(* CoDeSys 2.3 project: cy-wg-020-003.pro *)
(* Title: cy-wg-06 - ClevergyAS *)
(* Author: Andrea Ravasio *)
(* Libraries: Standard.lib 2.12.10 14:48:34, Util.lib 26.9.14 10:12:46, Visual.lib 2.12.10 14:48:34, WagoLibIdent.lib 25.2.13 11:12:16, WagoLibStatus.lib 2.12.10 14:48:32, SysLibFile.lib 2.12.10 14:48:34, SysLibRtc.lib 2.12.10 14:48:32, SysLibSockets.lib 10.2.11 09:20:54, SysLibEvent.lib 2.12.10 14:48:34, SysLibPlcCtrl.lib 2.12.10 14:48:32, SysLibCallback.lib 2.12.10 14:48:32, mod_com.lib 2.12.10 14:48:32, SerComm.lib 31.5.11 08:54:36, Serial_Interface_01.lib 22.4.13 12:50:14, Modb_l05.lib 22.4.13 12:50:12, Ethernet.lib 2.12.10 14:48:32, MBus_03.lib 22.7.15 16:25:47, WagoLibModbus_IP_01.lib 24.7.13 15:05:58, WagoLibMBX_01.lib 20.3.12 16:32:40, LON_01.lib 22.7.15 16:25:47 *)

(* PLC configuration (modules and I/O channels)
0750-9999/0545-0008 8 DO/DI Generic [Type_34_8_Channels] node 0, in %IB40 out %QB32 {INTTypePAAssignment = PLC; INTTypeModule = plugged}
  VPN_ST2 AT %IX20.0 [BOOLOnX_I] Ch_1 Digital input
  LAMP_AL AT %QX16.0 [BOOLOnX_Q] Ch_1 Digital output
  KEY_QE_ST AT %IX20.1 [BOOLOnX_I] Ch_2 Digital input
  EV01_OP AT %QX16.1 [BOOLOnX_Q] Ch_2 Digital output
  CTL01_ST AT %IX20.2 [BOOLOnX_I] Ch_3 Digital input
  EV01_CL AT %QX16.2 [BOOLOnX_Q] Ch_3 Digital output
  CTL02_ST AT %IX20.3 [BOOLOnX_I] Ch_4 Digital input
  EV02_OP AT %QX16.3 [BOOLOnX_Q] Ch_4 Digital output
  EV01_ST AT %IX20.4 [BOOLOnX_I] Ch_5 Digital input
  EV02_CL AT %QX16.4 [BOOLOnX_Q] Ch_5 Digital output
  EV02_ST AT %IX20.5 [BOOLOnX_I] Ch_6 Digital input
  AT %QX16.5 [BOOLOnX_Q] Ch_6 Digital output
  CIR01_AL AT %IX20.6 [BOOLOnX_I] Ch_7 Digital input
  AT %QX16.6 [BOOLOnX_Q] Ch_7 Digital output
  CIR01_AUTO AT %IX20.7 [BOOLOnX_I] Ch_8 Digital input
  AT %QX16.7 [BOOLOnX_Q] Ch_8 Digital output
0750-9999/0400-0008 8 DI Generic [Type_1_8_Channels] node 1, in %IB40 out %QB32 {INTTypePAAssignment = PLC; INTTypeModule = plugged}
  CIR02_AL AT %IX20.8 [BOOLOnX_I] I 1: Digital Input
  CIRD01_B_AL AT %IX20.9 [BOOLOnX_I] I 2: Digital Input
  CIR02_AUTO AT %IX20.10 [BOOLOnX_I] I 3: Digital Input
  CIRD01_B_AUTO AT %IX20.11 [BOOLOnX_I] I 4: Digital Input
  CIRD01_A_AL AT %IX20.12 [BOOLOnX_I] I 5: Digital Input
  CIRD02_A_AL AT %IX20.13 [BOOLOnX_I] I 6: Digital Input
  CIRD01_A_AUTO AT %IX20.14 [BOOLOnX_I] I 7: Digital Input
  CIRD02_A_AUTO AT %IX20.15 [BOOLOnX_I] I 8: Digital Input
0750-9999/0400-0008 8 DI Generic [Type_1_8_Channels] node 2, in %IB41 out %QB33 {INTTypePAAssignment = PLC; INTTypeModule = plugged}
  CIRD02_B_AL AT %IX21.0 [BOOLOnX_I] Ch_1 Digital input
  CIRD03_B_AL AT %IX21.1 [BOOLOnX_I] Ch_2 Digital input
  CIRD02_B_AUTO AT %IX21.2 [BOOLOnX_I] Ch_3 Digital input
  CIRD03_B_AUTO AT %IX21.3 [BOOLOnX_I] Ch_4 Digital input
  CIRD03_A_AL AT %IX21.4 [BOOLOnX_I] Ch_5 Digital input
  CIRD04_A_AL AT %IX21.5 [BOOLOnX_I] Ch_6 Digital input
  CIRD03_A_AUTO AT %IX21.6 [BOOLOnX_I] Ch_7 Digital input
  CIRD04_A_AUTO AT %IX21.7 [BOOLOnX_I] Ch_8 Digital input
0750-9999/0400-0008 8 DI Generic [Type_1_8_Channels] node 3, in %IB42 out %QB33 {INTTypePAAssignment = PLC; INTTypeModule = plugged}
  CIRD04_B_AL AT %IX21.8 [BOOLOnX_I] I 1: Digital Input
  CIRD05_B_AL AT %IX21.9 [BOOLOnX_I] I 2: Digital Input
  CIRD04_B_AUTO AT %IX21.10 [BOOLOnX_I] I 3: Digital Input
  CIRD05_B_AUTO AT %IX21.11 [BOOLOnX_I] I 4: Digital Input
  CIRD05_A_AL AT %IX21.12 [BOOLOnX_I] I 5: Digital Input
  CIRD06_A_AL AT %IX21.13 [BOOLOnX_I] I 6: Digital Input
  CIRD05_A_AUTO AT %IX21.14 [BOOLOnX_I] I 7: Digital Input
  CIRD06_A_AUTO AT %IX21.15 [BOOLOnX_I] I 8: Digital Input
0750-9999/0400-0004 4 DI Generic [Type_1_4_Channels] node 4, in %IB43 out %QB33 {INTTypePAAssignment = PLC; INTTypeModule = plugged}
  CIRD06_B_AL AT %IX22.0 [BOOLOnX_I] I 1: Digital Input
  ALARM_PB AT %IX22.1 [BOOLOnX_I] I 2: Digital Input
  CIRD06_B_AUTO AT %IX22.2 [BOOLOnX_I] I 3: Digital Input
  AT %IX22.3 [BOOLOnX_I] I 4: Digital Input
0753-0648 LON-FTT [Type_55_1_Channels] node 5, in %IB0 out %QB0 {INTTypePAAssignment = PLC; INTTypeModule = plugged; DataStream = 1F8B0800000000000400ED5DFB6FDAC8B7FFFD4AF77FF045BAAB560A0D06421E9B6445C134A83CB206D2ADDA0A3966006F8DCDD78FA4B97FFD3D33631B1B8F5F3C9286585A75893D3E73CECC99CF79CCF1F8F2AF5F0B957B4086A9E8DA5581FF502A704893F589A2CDAE0AB6352DF2B5C25FD7FFFD5F971D5D6B6B1632A692; DataStream = 8C387848332F7E99CA55616E59CB8BE3E3C7C7C70F8F950FBA313B2E974AFCF13FDDCE409EA385545434D392341915BCA726C94F15B85B439F19D2A20D8DCF4B17A5D2C529FC7B7251E22F4AB58B52157E14B87F94694F5AA0AB82A0A205D22CC940E38EA468CA58289D17B80152A74D5DB6C92D0B046CE80BFCFBAA509F4C; DataStream = B827DD3638995EE1E6C800067BC83674ADA5188B472075E78DCA39E96A203DA05BC99A5F151A17DF3F29D677F9A958E2CF8B8F33EE5D5782A1D1244E541E74D542AA2A7142A9FAFE7BA7DF2B705D7D62ABA8672FEE9101D40A309C1C8707B42B193FFBF7FF22D932C9B5F5ABCE45B83C448BA50A7DB427C0AD325590E1DD83; DataStream = BB78ACDA93EB528963FD7779ECDCF73D3190F525BA865BF487EFCE67F484AFE3FFF9AEB6B509FA75CD5F1ED31F1E5FC7318C794CE339BA1EB46E879A3E4154B2D583E4A6F708B369B049DF50668A26A9CCA6819BDE236DB3A3CB3FD1E4DA326C0432B87FFA1A74256D2259BAF1E4B5595DF135EB2FB11E49EAF554524DD2CC; DataStream = BBE2B5EA223CD174BAF15006FEF65A392ADBD06D503F5849179AA25E1570E705EED83720C87AD48D9F7792A148F72A32FD93B276CF772B496336D39A78CDF1B4E7BCBCAE3E3E15C237833A94A8470C5DEADD0DC7FAFDBF6303FDC746669436AD344A7B5044B769B8494069FC4D99DA944AA33268557ACD0A6B171FA15DA465; DataStream = 3A0DA344156D80B4C9505990A9F5FF196C27FD0AB4F3FDB9DE4E4432521E90AFA9FFCA9AF0B786A21B8AF5B412DEBB12683940C68322A3E113685E5DFEA9E98F2A9ACCD004B4D17727F048533100196020AFDBDAD286495D5D08B20C366FAAC8786EAE7BBA064CF8AF049A36746DAACC6C83D81458254B64580A32D707B56D; DataStream = 7A5DAD29CBFAF5C0631F9F2C3450FE0F5D572E8FBDDFBE557F1CBDEC7F5B44A8C4214265978800BE86659B2900411F382D13F1C06BF9DBC341398783F470D0B7ADD78507B583C183D3383C38DD191E4C15156117218D7BD082B6226E9AEC1E784D7788079EA22703824B32051E9CE47870B8EE015F3E1C3CA8C6E14175A778; DataStream = 90DE41C0EB1C9BFE342EC2AAED6F0F0AB51C140ED849289F1E0C2A9C87D250748468D450DA292A2CF53490404CFFAD9E26685835FDED01E1340784C3F512B2060DA13BAB8C6322CB97C7ACECF56629EDF80475918FC8501733A6A8C9A2BC530CCB96546E6A6B325D2DDCBD0A83BA9E79CE94468E59AB791E391DFEFF7E7964; DataStream = 68EE2487F9441B10269EC21278EAB0435390258314A566A4656E0BB8DFCD39F4C4CB53CA74845E2EA50CAD69A238033498E933CB3932BC226478792F3123301C4E6EF92C2E9774B6B35C9205AA8597EF62990618B0220E505AA7C14F3B4786C34286D7E7331C4E42E9EC2C0E1ACE76050D922A198B34A850C70D5362824334; DataStream = 8783C3828357E72894CF7338D8271CA4F7127244384844787D0EC22141425C56E16C6759051CF6A354C946F509E714504A4870E8E690705890F0FA9C84830104BE14E72490BBBB8184F983248F17FA24152C346FBE8C619233A4147CE47374382C74787D0E037F40F070120B0F273B4B37C29571AA5423C686BA6CE18669D3; DataStream = 8D0EED1C180E0B1872B721C785202E80BF70AB2B5AEA7D881C180E12185E9FC79023C3FE9121F718DE3C30E41EC3CBD533C5C1C2F9CE50C17C542C799E06151AAD264605414B9B7B7428E798705898903B0B39280440E1530E0A6F1E14724721DF91A08314F416F0A644BE23F1D6D1E1F5B90CF98EC41EF30B181BF2E4C29B; DataStream = 4785DC67C84121E430E4DB113930BC3E77214786FD2343EE31BC7960C83D86FCEC053A48C1B317CAF9D90B6F1E1B5E9FD3909FBDF00C672F648086FCEC85C3448657E735E4672F3CC7D90B2991213F7BE17091E1F5F90CF9D90B7B7DD93A2526E46F5A1F241CBC3A47E1905EB4FE1DE120BD979023C24122C2EB73100E0912; DataStream = 7ED3B3175242427EF6C24142C2EB73120E06107ECF4A47DFD90B299121AF743C5874787D0E435EE9F83C672FA44D37E6A50B07090CB9DB90E302FBEC851C18DE3430BC3E8F214786E7397B210786370D0CB9C790BF661D3A7B216DEE317FCDFA20312177167250089FBD9083C29B0685DC51C87724E82085CF5EC87724DE3A; DataStream = 3ABC3E9721DF917886B317F2E4C29B4685DC67C841817DF6420E0C6F1A185E9FBB9023C3F39CBD9003C39B068683F7184277CCD5AD249E2F8F3BBAD6958C9FFDFB7F81357275ED9A797DF93FDF1ACDFAB0FEEDF2AF5F0B957B408609D4AE0AFC875281439A0C03A6CDAE0AB6352DF2B5C25FD7970DC992547D767DD95254C4; DataStream = B54DF89F850C3481470A5C136EDE7924AA98066E86A7F0AA80FF85BF756321595EA31A6ED395FED50DDF7305EE56B2E65785C6C5770C5B86B420644CEEDDAFB3DAFBEF20C2171812F33BA6687E1F0CEBBD665D6C7E187EBD852709CE5D152280B0C089680AFC6A328A6D45DEC7C42F58023FE563BE725C2EF1658E3FBB2897; DataStream = 2EF872E17A1DAE092BCCABDC47C9744660002B55B6BED57E1438B28441FC0247D0F3AA705A29701896AE0A64609D2321E0DA83451FC63806120AE3C1501C35865452181A184D45A64F12AC9BC2E3F844890287B50CB35FE0469A029DFDA15A7FB6B5074955269C691930B1D08DA9DB868CFE98597FB285F2B12F68F68273C9; DataStream = 63EEC6169EBB5FCAC25E10510064E8EF22EF0A2346CB21F4465D96149EE80365A6398AE588E24A32F50D11A7C1536681C3DC21BA189C213DC1A09820D34833492FA05333980BB3AD5968860CD257DB1CC8F81D1AF2C74ACE9393CA892B1EE98925DCA837687FEA09CD71A7DFFB54E0FAD3A9892C42282CB04289E0CE50DD27; DataStream = 6E3920AED36ADF123990CEE1578C759B397111B255D89349C88D3D72D1522E1455554C24EBDAC44C2527CCF4B7CA6A2D790BA8095A01561E6B02274D26A0E3265B8C76BFB762FF84C5FE046BB94783327CE232ECE290D749CAF55F5EF15C7679AE53129C851F03E0B58CA7B8B51FCB3466C772B9ADB8DCB27A48AB4B83B98E; DataStream = 29A651A64AC58703954A483E620462746A70D3179304A444429AE4C1C359F15EB138DB619E03C4A30ED27E574E7080958CC850DB0819F85A94A8EB8E0371A336B14F8E69B1EF356415357D82E2D6542AFD34B5E8A56432FAD98396F23E25E55F938E7E542C6F72D60472C04F5F488AC662FF637BD84AD0B789F37034DBDE44; DataStream = D1A699AD1277CA1111E01F9F4D74043AF50B543E7545EA81326C2890461E8D1687E8994622AD2C42544342543D21AA7E217C6615F09693719364514ED99694D884185988189C3EE5705305A533A21B4B343424CD9448C8439C052359AE33E642F935761E8F168D3480D183C9CA0AE61940A17C721284BB2C2070CE443A874C; DataStream = B464B4855F05B700EED31FFEA54459F864E8F6726BC89E2DA3217B16E8616B004B42E1A04A6D84BDF7BAAE2249DB076CD5562A047D6EC8BF491E4D01C274E869F3376F3A281F23CD36A1ED5441EA6443516C42224E94A4483A3725B9290900F0D6966446A96CA7926CD3B289C1D9CCE57600DEB6E6785340A611BACE449CA8; DataStream = C1E14BCC8817488EF558F4C98EF99BC8E6E6B8B34AC5CC0B2D815806A9B6701CAA3FFC2BD4CD48560319497A12E5A60949F769277E3DDD7D4E92F6104849F23C3327398894242A25B9E23E3623499B4527246BFB4F42F43CE4C61C45E4BDD2A726A92118EBD3B1432E3A15E118A47D0B38402A922D62E1D5F8283D4576D274; DataStream = 888D29B19D656071663226CBB76936529A181E673BCBEA3B10109148950D6569E94C839C2A7098F848EC9AF3BA61484FDFF8DA0FACEE2D3A43539D93F0650ED1ADD295C78BB75A4CF2880FAFBDA75802D645B1FE35413E023D9480830835573CCA07B0C6D738792E19E0E02023459298AC8E063C90D2F66030F5A15CF92C24; DataStream = DCFA9030E6922E99C64D5D5C095C66DA5A4FE26FFCC98FB53513858E34D9551F34DAEDD5506C6EB4483F7FDBD224A533C6574FAB67955AF53429367386E1EF51BDE91B0626323262B435E9AB9E917EB23279D01B22E330296D1904C47296D039F59ADDA92392089AA9B7437CDB37E7BB851F8A3E3474E6DACD08F461828FF7; DataStream = D0A6E04303E9B13271650B634F8DA3DAB7DF182752FC6D1D7B4FC26F21AC49974D7FA6E0A6B636122AD266D67CFB10C091DF25173D00428FE3ABE7A5B322EFA657DC677EBB4C292E48D84DAA74F7715CF2A643A4544C0733EBFE4396087D0B98E57D5B7CFCAA06E5ACE20F9110F700CE71BCEF1711F2916306199B95D88556; DataStream = 1E94892DA91C5EB0649DEE20674CD9C5144BD1A9A330AFF04069373983E8C46402BF7C467EF9FDF05B4ECB6F3923BFE5FDF05B49CB6F2523BF95FDF05B4DCB6F3523BFD5FDF07B9296DF938CFC9EEC87DF5A5A7E6B19F9ADED87DFD3B4FC9E66E4F77487FCA6E3F02C3959CF746DE0D9B31706DFF3CD593F7F611CE6630C5D; DataStream = 12EFFC9E8C5E6A50E663AC5E22F37BB280A9119A8F318189CCEFC91CA6866B3EC61E2632BF27DB981ABBF918E398C8FC9E0C656A20E7632C6522F3A9ADE6CEAAFEDC88C0CBC2E082788E7C7268837860F5BD22977B6F03E80949C611B7D0356B7EC44DA4A7236EAEDBF88AA2D9163AE2684170CAAC69FACC59A584ABFC199B; DataStream = 435F91C48E78FC39B4B0984FE4B1B87460D92F71967460A6F8D515A38B07344BFCCA0CCA17944AB4EE91067B12A6B24A9449CC62E828519891F8448AAD7880DB7B12A3EC05D537A0D859E4A8B2E4981322D182E0FB7B92E4E4DCD32EB238B7AE915D386462F48BB4D8BB3C030A3219E461160E39581597C3F2BDDEB04DFEC6; DataStream = 9727E7573BF667DED60FF952CCE65BF6E4CB311E70ED2563DED19DFA8F0C0973F799987C795820D57BE86573E451026FB9865CF1B225C8B1C05BE7C737DCA7A2AF1E466C7B64793B422784E8F647E486156D947AEF9ED49310F51FE3ADB0403949A51CF0182AC1C566456CBFD19A92D8BAB5557F719BA892D74D7485C9695A; DataStream = 11974EA1D258450F484D5335E39536912792256596B105BB8D937619E82E5AE2B3677AC90F0345EF2E4B3D0D73438BE8E1D8D2C71867E3F4565975CAC9926D62B0756039515E8AB35582B37738C51E01B25516C8DED1BDB3C41D49F6368EB3F3B6B603EE416DF559A096297386AD1C26D012C948994C4C28F6BCB04A8398F8; DataStream = B8254A3B9988CA88625E41E8C23341F575C62E3C13365F61F0C22E1E7AA5D10BBB04E815872F65F61E7CA6F865D768767EEE9B21EF55F02C154DCCC07FE1A7B5B3B7CFFD2696FA7FAAB2000F3B83A1F53D96C2DCB2CBB5A8E7E8D07859A31B330A19F432C63F26A4B733C05B84DCC1725EC7F93CF7CC2FA9B55CEAA612159F; DataStream = A6299287E74351EA129F7F868C23B79E67FFC591229226C75FC0F7C60291CE134B2519AF183D8E97564246D4D354525D8DA76EF59EE2FE8FB9F0844C51AB15C419665E0E048EACD2F24066F55ED5AA2674E73AE939524EA0BDF95132103B8F7DA7B1048E9368378F3CCABF51C2E019B3040E61D65938E52A33844E9E906008; DataStream = CD34D2C16EE342683DD05D74088D23D52D15D1B779545EED1E9D57D624DF3821893531F80A51CDAF88CE8B3753559AA5377307A38D89C51A4ECEB6D86E92214ADE88642A9E42A9B079DFC1562A9F4E08579D7720C96A0D3D7F294753313191C936724C1C1A2F52CED1B7ADA23E2D12AFCCDC460ADDB6F00B6694D08B1477F4; DataStream = 97482BCA8A21DBCA567AA5039DB143E7450A3D9C3931E9C9893B981487D28B147E74913C9734053A2E4E255BDD6A66161EAD31A1F522C5202D8426F792FC13C45154DBD86A7EA60EADB143EB99CAFEFA0FC8281A92364BCB3C3324D781CA985079114B3202BBBA03296C4C669F6224581001BFBB6A645E1F4C5990476B9FEB; DataStream = 23C1A28C344CA368E9C50592CCF40B2462763031BCD3E2107B11CBD2D0170B5B738E3A30332E7CA65C3250DCC3A24F6F635AD0379A808D51A7452BBD23C61406CB31C694C6D6DEFCB0A4F242578EA2A2159798437CF8D0163279E28C156DEC127C117B434F222E8229DF461E955019B30FEFDC878DE94A9A0D9826EB9A65E8; DataStream = 6A4AD699399905A1347628BD50D4B2049F8C6EDD6F2109A8925B93F3FC8686CA808DB6A14CD2825794182E9917B130225AEA86555C48E6CF6DC43008993126F32256C5E548D16645FC81AC6D6459AE68918F6DBD884DF10B846DC2AE04C2B45EC4AA90CD90A2A65BCAF4A938C916EA33A5A25B2094E078BF717F82551191C9; DataStream = 7EDF37D5C2817B80C78BA58AE2774E3738A2EF8CF39B16AF1412F7693CA0498AD736985B6CBEE7F771FAD61689FED53BD8E4239A1BA4554DE7C1B5FC232975A15955B4975DC355D94A64B5D1FA0E6174A9913329EE3B121F69C67D6D82FE971C8964ABAA5BBE96A857836DCE140E1E361577D6C87AFD47D4F15309878D7882; DataStream = 92B6E47CBB2DCF5771D2E3EE16C149CAC297F2692D701E4DF9B4C27B5B8BF8932D78EF81C42E99DFB1F07DCA253818EEB497E35EBB9820F0C491C935906A2A769A2D46B2CB43BE4269F906E22CA0C8CC39BFB9AB37B845C4010251678C05BF791937C51EF9982D9D6AE4EC9BD797BEF6C1BFB8D5971386D2CC39EB67B5C175; DataStream = 7D492BEB020979CE59C261895AE2B837EA1438517A246DE8101D07A90C3075CD522495936419C75E06C27BD74C72FD5BA1371EF6C703A1D74C41E911EFEF2690128586D0BE13FC5C86996CA8BA8938490370971E9073F418936CA3D31F08E356BB13A0588EA13841D81626D36C0A1D6118265D099116C9919DC0E6847C9246; DataStream = 379EDCEF0930A937DB3004C3BEF815D65DFFF3E8D64FBC1A260E2CEB8B8C533516EB7EAA270954334CDB1A657AC0DEB14FA399EA5DF3ABB7776E6056ED1EA4D06E521662E1E34DA7C8E04C9B0808662882E03F2D0144FC1C22D3F46652D5F59FF8C8DF244A742E09AD38C5160C4337387C0AE71269D86B8954C3011DFA56BD; DataStream = DD89D76C8FE4648DE9784E05518C57EBE0502A1AB7CAAD448FE5A8D714C42FB88E2A4EA93D96B13EC3281C630D4C188D767F9DE5B05A0759C62F414E38924761521CB6BB427F345C275B0B91FDA2C06A79E44C827732E210663F82E89776AFD9FFB24EF3344473ED50562FC1C8245A1F0D6FD6499E8549D2D54C0D956E81CE; DataStream = 2E71D88CD88801541B0D61308029ABDFAD29D9790260DCA3271D9054E8334F4500D20341F83C6EF7EEEA1DBC6DEF5B10A5F09C39ADBFD4DB4CAF3378DF478A4F873DA70EF604DE3109B2305A4EB00FE7CDEF1CB4123127B8DE19DF087550F1200C8517CF3AC9A9AE5B91245BFDFE709D64789D37D1BD3D23C70BE20F7A6109; DataStream = DFE1599634FA9AC2FB08E24DE1E3E85390761896DA3EAA36653D15F176AFD50FD20E4FF0E0C9041F323BE383AF83A1D00D77115E9FC3B973B634A7989C536B104114347224B034B31846930059095C7C0D4C97E61CA2944E8646BF87BF961650DC62180F714F1344B690A12B7D3A55158D890540B2DF6A75DABD804B520CEB; DataStream = 1F2D0EC5C5B50A9D540D7FE90F467E213DC1F2E526D0D2D28954BE0D1317863840E7B9644C1E25BC7742AF458938EA7DEEF5BFF402FC8495D7B5EEBE77AA9C6194D63825C8B54432FE86E524AAD36447A0A773EB949738B3A031AD0126D9C7B3D56C0FC9B1B0EBCB59F358CA48B6DEE9FAE9C6F90643DD92D463B796801482; DataStream = 3E60DF9AF4C773EF701A47D7A02B526106C6DEE4DCC6305FF80C3A0B6912A04DD4A80DFBC3F1E0AE4178E2E39D8A585E981BE46BF4CBF1CE452C7DE6B6C81AFD4ABC87E1144783D5760AA4E9A4A948323866C80FE43B60B73BDD21B8FF627078C2D010473E6A74FCE4CBF10E07253F5766F30CECDFB43FDDB0F967781F711D; DataStream = 440910E8A09CE08B30072869E4438A197644D88493C63CA4910C3B15312689C31D629A615F2368278E7498EFF0526D0112AC835294A3D11631C9004196E30F0401D58AE989DE8A428870785162C24503E18F0D4FC04DD7ED7B70D7DF91FA87F7A9BA198A1F03B8CFB342005F1FE00163843175F2FD0E17B0DFA10FB30F4760; DataStream = 640C45FBA942A08011DC8C3171B8EBC1E8F62ED07578D506C5C33BDCC4154F3F8A4361300C0D6378F146F4936DC6485FAC690BAFE5407F0B9A8AE390F6A018BA86DF3701DCC6A60969267522E80BC410DAC97376ECE1B020F4EE1AFDEEEDB85BFF27C04178D1073890EE35EC48AA603596B6954AD86EBFD71EF64562880376; DataStream = 8F118E0485F56C2A4C2332A28C3CE9A3DEEEE1D913C480B75766E428F0177D3969B9545DB72B32A0C4B4EB43F81782BF7E305E0FB3DE8788D2A0B41247254C2FCC27A5073E2049542451FC52177BED5E20D2A894D38568674E88167A473E6386E8364DFEB3A33FE2221ABA52966BEFD8336976843BA1330E8FB7778B6922FC; DataStream = 77E3BC3EAF1DD318F8EFC6F96B37605A3612AB12EFA7759429E206D21401316217882533B9771FEB0D7C38B077484199099EB76B9E48D826DCD2EF683FA5EAA412D54939DE5D2344073E6340ED71887E358A7E25DE5F23F487D4A01DB7486DE0BBA6622E55E9E97DB89793A85EAAF14E1BE9E516E089707FC4916D8906CE9C; DataStream = C980270284044B0CC751C2D5A2BAADC5BB72A49BA819398B227A16EFC645F12E0E7B475407E057DC20F2A548852B25387AA46F425EA558E02E17563791A3C6D7183E5F22D4617608D6855E66CA8875E2DF29B04E203599CE8B5364F3C3400BFD01AE7845416CCA7DB15BEF30B2E2A68F5EC4B3CDF6A0FEB12334E3518F1606; DataStream = B99CB96F1A31098E6E9BF521DE59AF0F47837814BC45064E327964DD52C308CA03A1D3228E503C063AB93C2970C4531CABF54E5DECC6C39E23BFF31E153E2A88163731C98AC26D5F1C828731F81C8F737DB7642C7686FA7760FDDB4D211ED302BA134149E8E1A98E472DD1D1383A25098A2776EF98EC8551A94142D534FAD3; DataStream = E8087591A13E61500AD074CAFF624886A6998135CE2852DD21D5448A7B3A169332A109EB6FD86E7D7586B7C9C019D6AADCAC0FE672656C320590644AF24DB8D693F36A3D995D75EBBD114E830EC560DC165E64E10E305491CA8AB80E44A1DB871517EA80B1E7443BF055ABE10A1592D6A3624C9599ED80F5923A25E43B8CCC; DataStream = 6E6FC5FE27B11E9CFCF072A4FA446AB08A6E0D16A949E3DE050BB39836C6D333511808C1AD0FC66AFD85641BA8D3CEBC6D0790307601874987173095022050E2547D16CB69A71FF0FF19B164479720669D7BF3B04AF5E21DC641E376886FD06F8E4574D5E9D79BCC0960EC5AD91AE94CB60D03BC0B15EF8C4A13E8CBE9FD03; DataStream = D79E06B879944C6E2EA934F6C3FAAD3E1D4103C5E41E1515C7B4265874CEB035BA776BE80BFA387E6D1FA7EE57CF7F881AF1518FC53C2312BD013A09DC0F3DCE964ED55C706C49691236FB12FECE3BD50AF0B1605470DA1FDFF08BE57F9488F608F11FE2C036258B7553EF0C9972B14C3FF065C48BB61ADA7B3453C868470E; DataStream = 28D8EFBAC8EE3C8C63234D753530AAEF28DBDE8B52BC3203CDE8723449471AFA65E1A5435C5D7DE97A84EFF0268F53F4877DDF23580126293F84BB47F401EE1EBF0D70C4214BFEF01EAFE6247D589FFC850DFEED3DE2FEF88FAD5B7F2A1315D15F78C780FEA2F3EA5CC55B42B28C9616557A474B8E381DA7021E15936A03D6; DataStream = 19A0A9CC34DD009508746B20CB3634135362D07734726AE144051923F245D269A0BB286F6D28DC3287BF9AD2F5AE3AAEB75361C676B81FA21C6E1C35A470B91BD45CE1B4A2645B3A218061047F864D9B21BC776E3D22A405F23F387FC73435A4D3FA68D80FA3039248C584AEA9CC4223F2E48D501FC6FBE1F5151745078A65; DataStream = 6087A67C1E714D35BB8E8490EF8ABD4FE32F623758C3C4A8BDD2753591D746BFDF89F7C399BC6ACA6C0E119C6DCC6266ADFDE9060062247E12E2BD72660F38AF2AEB6C0F8490C759D475EE19CEC04A31F016A7E3D6D071B1ADA56D452B40BFD54AF0D5BDF8F91E618238E661A75E09BDF590276CF305583C33F0209E702D84; DataStream = 454B4ADE919F4B7BB164BA2B84B2D015C44F21B5636C0F29DE28D0A4220290994A60AD013C70D10ED377255DB4EABD71BFD7F99AE0CA3B2AF7A85873929DC6297E9D76EA98EFE81E44213CA10CDFBE2DA3E242FA89BBA115A411F4DA0D21C18577EA5BC9602792EBD6FF092F6C86C70E63AB2F407F31521CE3F188272B34FA; DataStream = BD7EF76B829BDE44737BA14CBC10239E6653B81975D72A80C2ABAE01C07B6FA420D7A877DA1F4588B013FCEE95F6CAC962138D0DCD36638D7944616D81A14B41152C563D6933C79B52CA42CC9C877864A7EAC637770DE223475B05AF41ACF34CA1B31F4FCBBB1F726583F6F83858027D8C2BF5AE2F49BD5EDB84FF8143E0D4; DataStream = 5E3721D0B84386090DB1B67C006AB8192DEA6E2D212A68913A22AFCD096ED295FED50DDF63C0B064CD41B72EBE3B9C132A26F7EED759EDFDF78EAE7DD18D9FE67752A0FD1DD7E834EB62F343EBD6A9416B0333A512C7FA0F6445536017E2ABD856F8030E03FC0906BC3C8FF9CA71B9C49739FEECA25CBA80F50AD2DB1AF1F5; DataStream = 24157A249F7B665CF3BC17B7D61D7F278FEB7B419DA2C9CA5252234E2D188040F893774EFB50013E0C7E173C2E09578DD2F70A103E308B7ED4DAD7E9FA414AE19EB4074574EFE241F51D8E15AEFB4FE876FD40ADE8F48EF6A0BB1F17F7775A61761AECC47B99872861BC64B8094817E8E4344D27B54027B172E01658966027; DataStream = D5149D9C063A599D891729CAADBE365ECE8A0D291FEBDA6AF51E37F046A63EBBFEF103FEE8E0772160194F25195DFF3F0534515341320100; DataStream = .; DataStream = .; DataStream = .; DataStream = .; DataStream = .; DataStream = .; DataStream = .; DataStream = .; DataStream = .; DataStream = .; DataStream = .; DataStream = .; DataStream = .; DataStream = .; DataStream = .; DataStream = .; DataStream = .; DataStream = .; DataStream = .; DataStream = .; DataStream = .; DataStream = .; DataStream = .; DataStream = .; DataStream = .; DataStream = .; DataStream = .; DataStream = .; DataStream = .; DataStream = .; DataStream = .; DataStream = .; DataStream = .; DataStream = .; DataStream = .; DataStream = .; DataStream = .; DataStream = .; DataStream = .; DataStream = .; DataStream = .; DataStream = .; DataStream = .; DataStream = .; DataStream = .; DataStream = .; DataStream = .; DataStream = .; DataStream = .; DataStream = .; DataStream = .; DataStream = .; DataStream = .; DataStream = .; DataStream = .; DataStream = .; DataStream = .; DataStream = .; DataStream = .; DataStream = .; DataStream = .; DataStream = .; DataStream = .; DataStream = .; DataStream = .; DataStream = .; DataStream = .; DataStream = .; DataStream = .; DataStream = .; DataStream = .; DataStream = .; DataStream = .; DataStream = .; DataStream = .; DataStream = .; DataStream = .; DataStream = .; DataStream = .; DataStream = .; DataStream = .; DataStream = .; DataStream = .; DataStream = .; DataStream = .; DataStream = .; DataStream = .; DataStream = .; DataStream = .; DataStream = .; DataStream = .; DataStream = .; DataStream = .; DataStream = .; DataStream = .; DataStream = .; DataStream = .; DataStream = .; DataStream = .; DataStream = .; DataStream = .; DataStream = .; DataStream = .; DataStream = .; DataStream = .; DataStream = .; DataStream = .; DataStream = .; DataStream = .; DataStream = .; DataStream = .; DataStream = .; DataStream = .; DataStream = .; DataStream = .; DataStream = .; DataStream = .; DataStream = .; DataStream = .; DataStream = .; DataStream = .; DataStream = .; DataStream = .; DataStream = .; DataStream = .; DataStream = .; DataStream = .; DataStream = .; DataStream = .; DataStream = .; DataStream = .; DataStream = .; DataStream = .; DataStream = .; DataStream = .; DataStream = .; DataStream = .; DataStream = .}
  AT %IB0 [BYTEOnB_I] First Byte of 24
  AT %QB0 [BYTEOnB_Q] First Byte of 24
0750-0464#04 2/4 AI RTD / ADJ./ HA [Type_44_4_Channels] node 6, in %IB36 out %QB28 {INTTypePAAssignment = PLC; INTTypeModule = plugged}
  S01 AT %IW12 [INTOnW_I] Channel 1
  S02 AT %IW13 [INTOnW_I] Channel 2
  S03 AT %IW14 [INTOnW_I] Channel 3
  AT %IW15 [INTOnW_I] Channel 4
0750-0650/0003-0000#03 RS 232 C Interface (Adjustable), 3 Byte [Type_21_1_Channels] node 7, in %IB60 out %QB52 {INTTypePAAssignment = PLC; INTTypeModule = plugged}
  AT %IX16.0 [BOOLOnX_I] Transmission acknowledgement
  AT %IX16.1 [BOOLOnX_I] Reception request
  AT %IX16.2 [BOOLOnX_I] Initialization acknowledgement
  AT %IX16.3 [BOOLOnX_I] Input buffer is full
  AT %IX16.4 [BOOLOnX_I] Number of received characters Bit 0
  AT %IX16.5 [BOOLOnX_I] Number of received characters Bit 1
  AT %IX16.6 [BOOLOnX_I] Number of received characters Bit 2
  AT %IB33 [BYTEOnB_I] Input data Byte 0
  AT %IB34 [BYTEOnB_I] Input data Byte 1
  AT %IB35 [BYTEOnB_I] Input data Byte 2
  AT %QX12.0 [BOOLOnX_Q] Transmission request
  AT %QX12.1 [BOOLOnX_Q] Reception acknowledgement
  AT %QX12.2 [BOOLOnX_Q] Initialization request
  AT %QX12.4 [BOOLOnX_Q] Number of characters Bit 0
  AT %QX12.5 [BOOLOnX_Q] Number of characters Bit 1
  AT %QX12.6 [BOOLOnX_Q] Number of characters Bit 2
  AT %QB25 [BYTEOnB_Q] Output data Byte 0
  AT %QB26 [BYTEOnB_Q] Output data Byte 1
  AT %QB27 [BYTEOnB_Q] Output data Byte 2
0750-0653/0003-0000#03 RS485 Interface (Adjustable), 3 Bytes [Type_21_1_Channels] node 8, in %IB68 out %QB52 {INTTypePAAssignment = PLC; INTTypeModule = plugged}
  AT %IX18.0 [BOOLOnX_I] Transmission acknowledgement
  AT %IX18.1 [BOOLOnX_I] Reception request
  AT %IX18.2 [BOOLOnX_I] Initialization acknowledgement
  AT %IX18.3 [BOOLOnX_I] Input buffer is full
  AT %IX18.4 [BOOLOnX_I] Number of received characters Bit 0
  AT %IX18.5 [BOOLOnX_I] Number of received characters Bit 1
  AT %IX18.6 [BOOLOnX_I] Number of received characters Bit 2
  AT %IB37 [BYTEOnB_I] Input data Byte 0
  AT %IB38 [BYTEOnB_I] Input data Byte 1
  AT %IB39 [BYTEOnB_I] Input data Byte 2
  AT %QX14.0 [BOOLOnX_Q] Transmission request
  AT %QX14.1 [BOOLOnX_Q] Reception acknowledgement
  AT %QX14.2 [BOOLOnX_Q] Initialization request
  AT %QX14.4 [BOOLOnX_Q] Number of characters Bit 0
  AT %QX14.5 [BOOLOnX_Q] Number of characters Bit 1
  AT %QX14.6 [BOOLOnX_Q] Number of characters Bit 2
  AT %QB29 [BYTEOnB_Q] Output data Byte 0
  AT %QB30 [BYTEOnB_Q] Output data Byte 1
  AT %QB31 [BYTEOnB_Q] Output data Byte 2
Fieldbus variables [FB_VARS] node 1, in %IB0 out %QB0
Flag variables [FLAG_VARS] node 2, in %IB0 out %QB0
Modbus-Master [MB_MASTER] node 3, in %IB0 out %QB0
*)

(* Global variable list: Global_Constants *)
VAR_GLOBAL CONSTANT

	Plant_NAME			: STRING :='cySN:20 cyVER:1 - ';
	Plant_SN			: DWORD  :=20;	(* S/N Impianto di telecontrollo *)
	Plant_SW_VER		: WORD   :=1;		(* Versione SW installata *)


	(* Colour defines *)
	COLOR_RED			: DWORD	:= 16#2020F0;
	COLOR_YELLOW		: DWORD	:= 16#20F0F0;
	COLOR_GREEN			: DWORD	:= 16#20F020;
	COLOR_LIGHT_GREEN	: DWORD := 16#006000;

	(* Parameters *)
	Plant_DefaultTAmb	: INT	:=100;		(* [.1°C] Temperatura ambiente di default in caso di rottura sonda *)
	Plant_MaxRunTAmb	: INT   :=250; 		(* [.1°C] Temperatura ambiente massima funzionamento impianto *)
	Plant_AntiFreezeTAmb: INT   :=-40;		(* [.1°C] Antifreeze temperature, start circulators *)
	Plant_VRD_TAlarm	: INT   :=450; 		(* [.1°C] Temperatura di allarme VRD, blocco *)
	Plant_VRD_TMax		: INT   :=430; 		(* [.1°C] Setpoint massimo per uscita VRD *)
	Plant_VRD_TDefault	: INT	:=300;		(* [.1°C] Temperatura di default in caso di errore climatica *)
	Plant_CirOffDelay	: TIME	:=T#30m;	(* (Def.T#15m) Ritardo spegnimento pompe per ricircolo caldaia *)
	Plant_CirOnDelay	: TIME	:=T#15m;
	Plant_MaxWaterLoss	: WORD  :=2;		(* [lt/h] Massima perdita del circuito *)

	(* Filesystem *)
	FilesPath  			: STRING :='S:\';

	(* TCP Logger *)
	Logger_SERVER		: STRING:='';
	Logger_IP			: STRING:='192.168.100.3';
	Logger_PORT			: WORD  :=80;
	Logger_GETSTART		: STRING:='GET /cygmsrv/hsgm.ashx?';
	Logger_GETEND		: STRING:='$R$N$R$N';
	Logger_CHECK		: STRING:='True';
	Logger_CRLF			: STRING:='$R$N';
	Logger_DataFile		: STRING:='S:\LOG.DAT';
	Logger_DataFileOld	: STRING:='S:\LOG.BCK';
	Logger_IndexFile	: STRING:='S:\LOG.IDX';
	Logger_ConnRetries	: BYTE:=5;
	Logger_RecoverMsgs	: BYTE:=25;

	(* TCP Remote *)
	Remote_PORT			: WORD  :=10;
	Remote_WELCOME		: STRING:='Connected$R$N';
	Remote_OK			: STRING:='OK$R$N';
	Remote_ERROR		: STRING:='ERROR$R$N';

	(* TCP Sockets *)
	MAX_SEND_TCP_SERVER					 : DWORD:=3000;(*60000*)
	MAX_RECEIVE_TCP_SERVER				 : DWORD:=3000;
	MAX_RECEIVE_TCP_SERVER_SOCKET	 	 : DWORD:=1500;
	MAX_SEND_TCP_CLIENT					 : DWORD:=3000;(*15000*)
	MAX_RECEIVE_TCP_CLIENT				 : DWORD:=1500;
	MAX_RECEIVE_TCP_CLIENT_SOCKET		 : DWORD:=1500;
	MAX_RECEIVE_UDP_SERVER				 : INT  :=1472;
	MAX_RECEIVE_UDP_CLIENT				 : INT  :=1472;
	CONNECT_WATCHDOG_TIME				 : TIME :=t#10s;

END_VAR

(* Global variable list: Global_Retain *)
VAR_GLOBAL RETAIN PERSISTENT
	Mode_Manual : BOOL := FALSE;

	CAL01_Clima : typ_Clima;
	CAL02_Clima : typ_Clima;

	VRD01_Clima : typ_Clima;
	VRD02_Clima : typ_Clima;

	Ctl01_Counter	:	DWORD;	(* Water counter *)
	Ctl02_Counter	:	DWORD;
END_VAR

(* Global variable list: Global_Variables *)
VAR_GLOBAL

	SYS    : typ_SYS;
	Logger : typ_Logger;

	Lamp	:	PLANT_STATUS;
	T_AMB	:	INT;		(* Environment temperature *)

	(**** PLANT OBJECTS ****)
	(*...*)
	(* Boiler *)
	CAL01	:	obj_CAL_VT100GC1B := (ID:=1);
	CAL02	:	obj_CAL_VT100GC1B := (ID:=2);

	(* Cascade *)
	CAS01	:	obj_CASCADE	:= (Tmonitor_On:=T#45m, Tmonitor_Off:=T#30m, DeltaTempThr:=70);

	(* Water counter (NB: weight is multiplied by 10) *)
	CTL01	:	obj_CTL	:= (ID:=1, Peso:=25);	(* Domestic water	-	2.5 mc/h --- 2 impulsi/litro *)
	CTL02	:	obj_CTL	:= (ID:=2, Peso:=25);	(* Compensation		-	2.5	mc/h --- 2 impulsi/litro *)

	(* Heat counter *)
	CTB01	:	obj_MBUS_CTB_SHARKY775 := (ID:=1, Address:=16#51865849);

	(* Cronothermostat *)
	THER01	:	obj_CRONTER := (ID:=1, Local_MaxRunTAmb:=250);
	THER02	:	obj_CRONTER := (ID:=2, Local_MaxRunTAmb:=250);
	THER03	:	obj_CRONTER := (ID:=3, Local_MaxRunTAmb:=250);
	THER04	:	obj_CRONTER := (ID:=4, Local_MaxRunTAmb:=250);
	THER05	:	obj_CRONTER := (ID:=5, Local_MaxRunTAmb:=250);
	THER06	:	obj_CRONTER := (ID:=6, Local_MaxRunTAmb:=250);

	CronEd	: 	obj_CRON_EDITOR;

	(* Pumps *)
	CIR01	:	obj_MODBUS_CIR := (ID:=1, Address:=1, OnDelay:=T#1m, OffDelay:=T#30m);
	CIR02	:	obj_MODBUS_CIR := (ID:=2, Address:=2, OnDelay:=T#1m, OffDelay:=T#30m);

	(* Double pumps *)
	CIRD01	:	obj_MODBUS_CIR_DOPPIO_new := (ID:=1, Address1:=3, Address2:=4, OnDelay:=T#1m, OffDelay:=T#10m, Mode:=1);
	CIRD02	:	obj_MODBUS_CIR_DOPPIO_new := (ID:=2, Address1:=5, Address2:=6, OnDelay:=T#1m, OffDelay:=T#10m, Mode:=1);
	CIRD03	:	obj_MODBUS_CIR_DOPPIO_new := (ID:=3, Address1:=7, Address2:=8, OnDelay:=T#1m, OffDelay:=T#10m, Mode:=1);
	CIRD04	:	obj_MODBUS_CIR_DOPPIO_new := (ID:=4, Address1:=9, Address2:=10, OnDelay:=T#1m, OffDelay:=T#10m, Mode:=1);
	CIRD05	:	obj_MODBUS_CIR_DOPPIO_new := (ID:=5, Address1:=11, Address2:=12, OnDelay:=T#1m, OffDelay:=T#10m, Mode:=1);
	CIRD06	:	obj_MODBUS_CIR_DOPPIO_new := (ID:=6, Address1:=13, Address2:=14, OnDelay:=T#1m, OffDelay:=T#10m, Mode:=1);

	(* Temperature probes *)
	TPV01	:	obj_TPV := (ID:=1);
	TPV02	:	obj_TPV := (ID:=2, IN_WMIN:=50 , IN_WMAX:=800);
	TPV03	:	obj_TPV := (ID:=3, IN_WMIN:=50 , IN_WMAX:=800);

	(* Zigbee temperature probes *)
	ZTHL04	:	obj_ZTHL := (ID:=1, Address:=1);
	ZTHL05	:	obj_ZTHL := (ID:=2, Address:=2);
	ZTHL06	:	obj_ZTHL := (ID:=3, Address:=3);
	ZTHL07	:	obj_ZTHL := (ID:=4, Address:=4);
	ZTHL08	:	obj_ZTHL := (ID:=5, Address:=5);
	ZTHL09	:	obj_ZTHL := (ID:=6, Address:=6);
	ZTHL10	:	obj_ZTHL := (ID:=7, Address:=7);
	ZTHL11	:	obj_ZTHL := (ID:=8, Address:=8);

	(** Communication **)
	(* ModBus *)
	MODB01	:	obj_MODBUS		:= (ID:=1, COM:=3, BAUDRATE:=BAUD_19200, RS485:=TRUE);
	MODB02	:	obj_MODBUS_TCP 	:= (ID:=1, IP:='192.168.100.11');

	(* M-Bus *)
	MBUS01	:	obj_MBUS		:= (ID:=1, COM:=2, BAUDRATE:=BAUD_2400);

	(**** SIMULATION ONLY ****)
	(*...*)
END_VAR

(* Global variable list: LON/Module_1/InterfaceBlock_Module_1 *)
VAR_GLOBAL CONSTANT
(******************************************)
(* Automatic generated code, do not edit! *)
(******************************************)
	abSignature_Module_1 : ARRAY[0..15] OF BYTE := 16#67,16#E5,16#C2,16#E0,16#43,16#BD,16#55,16#4D,16#BE,16#30,16#A9,16#FE,16#D9,16#26,16#7B,16#E7;
	wConfigSize_Module_1 : WORD := 522;
	abInterface_Module_1 : ARRAY[0..130] OF DWORD :=
		16#302841AA, 16#214BDC0F, 16#6041B800, 16#06246830, 16#428B2E71, 16#64B95263, 16#FE000902, 16#2A050140, 
		16#0028C092, 16#037C10FF, 16#6D81026F, 16#0418B0E4, 16#C75C1D07, 16#9CD47157, 16#5A1D2B75, 16#1D531D1E, 
		16#4F0D2658, 16#5AC76C1D, 16#2D5F874A, 16#FE884D09, 16#CE34C958, 16#4CA0345D, 16#856A742A, 16#B26FDD52, 
		16#2BF66959, 16#74C79655, 16#966CD09D, 16#DFE60549, 16#2C48B975, 16#B66DFB76, 16#48BA6ECB, 16#955B162D, 
		16#B7300196, 16#2B35AD5D, 16#65EBC62D, 16#2106DDB9, 16#564CBE30, 16#DDA96F05, 16#AD4B372C, 16#255378CD, 
		16#36ADD181, 16#59D42ACB, 16#9B603585, 16#DDC49858, 16#EA45B329, 16#CD59F616, 16#B50A12E0, 16#56B5BE52, 
		16#8C890100, 16#5AAA1481, 16#B253E154, 16#6C831684, 16#A2ADDCB0, 16#4ABD13A9, 16#950B79D9, 16#4A948694, 
		16#4DBF5E45, 16#CA018948, 16#054C41E5, 16#B86DCB52, 16#2FBEA018, 16#40AAB4D0, 16#A1F866E7, 16#E288A8D1, 
		16#D192DBA2, 16#80E25047, 16#84B4644B, 16#B225A097, 16#59A9F8AC, 16#2D5B376E, 16#7B32E9CE, 16#B7AE3099, 
		16#2D551A30, 16#03F1D236, 16#C96176D0, 16#D94ABD0C, 16#94950479, 16#60B2886A, 16#25C9C990, 16#4CBCB141, 
		16#32D60DA9, 16#6A1D86D9, 16#514404B2, 16#129278D2, 16#09A12969, 16#AB6529E7, 16#90EE2F05, 16#10604094, 
		16#FE031C08, 16#418817F3, 16#84320FB0, 16#238F21C0, 16#6F23C08A, 16#003E98A3, 16#80677304, 16#10728E02, 
		16#0E02FC59, 16#02343A1A, 16#183B223A, 16#804705C0, 16#47864080, 16#47408082, 16#2E208347, 16#A304A014, 
		16#121794C3, 16#81595C58, 16#C785A471, 16#6820171C, 16#7201925C, 16#88CB8581, 16#5D283A17, 16#2378C120, 
		16#1724EF85, 16#0B5F78C0, 16#85687C01, 16#CE17B4F2, 16#814B5FD8, 16#F6856C7D, 16#E8DC173C, 16#6001805F, 
		16#047C0101, 16#97310112, 16#A061674C, 16#20841212, 16#4081A022, 16#2F7F96E0, 16#DE43C10B, 16#E9BB69D5, 
		16#D9FDA786, 16#FEFC5E93, 16#0000181B;
END_VAR

(* Global variable list: LON/Module_1/Runtime_Module_1 *)
VAR_GLOBAL
(******************************************)
(* Automatic generated code, do not edit! *)
(******************************************)
	mbxModule_1 : MBX_Full;
	InDataTelegram_Module_1 : ARRAY[0..255] OF BYTE;
	OutDataTelegram_Module_1 : ARRAY[0..511] OF BYTE;

	xInitRunning_Module_1 : BOOL := FALSE;
	unLastLen_mbxModule_1 : UINT;
END_VAR

(* Data type in LON/Enumerations *)
TYPE alarm_type_t :
(
	AL_HEADER := -13,
	AL_FOOTER := -12,
	AL_DEBUG := -11,
	AL_INFO := -10,
	AL_SYSTEM_INFO := -6,
	AL_VALUE_INVALID := -5,
	AL_CONSTANT := -4,
	AL_OFFLINE := -3,
	AL_UNKNOWN := -2,
	AL_NUL := -1,
	AL_NO_CONDITION := 0,
	AL_ALM_CONDITION := 1,
	AL_TOT_SVC_ALM_1 := 2,
	AL_TOT_SVC_ALM_2 := 3,
	AL_TOT_SVC_ALM_3 := 4,
	AL_LOW_LMT_CLR_1 := 5,
	AL_LOW_LMT_CLR_2 := 6,
	AL_HIGH_LMT_CLR_1 := 7,
	AL_HIGH_LMT_CLR_2 := 8,
	AL_LOW_LMT_ALM_1 := 9,
	AL_LOW_LMT_ALM_2 := 10,
	AL_HIGH_LMT_ALM_1 := 11,
	AL_HIGH_LMT_ALM_2 := 12,
	AL_FIR_ALM := 13,
	AL_FIR_PRE_ALM := 14,
	AL_FIR_TRBL := 15,
	AL_FIR_SUPV := 16,
	AL_FIR_TEST_ALM := 17,
	AL_FIR_TEST_PRE_ALM := 18,
	AL_FIR_ENVCOMP_MAX := 19,
	AL_FIR_MONITOR_COND := 20,
	AL_FIR_MAINT_ALERT := 21,
	AL_FATAL_ERROR := 30,
	AL_ERROR := 31,
	AL_WARNING := 32
);
END_TYPE

(* Data type in Logger *)
TYPE en_Logger_ErrLev :
(
	EL_Log			:=0,
	EL_Wrn			:=1,
	EL_Alarm		:=2,
	EL_AlarmStop	:=3
);
END_TYPE

(* Data type in Logger *)
TYPE en_Logger_Status :
(
	S_Logger_UNKNOWN := 0,
	S_Logger_IDLE,
	S_Logger_WAITCONN,
	S_Logger_WAITTX,
	S_Logger_WAITRESP,
	S_Logger_ERROR
);
END_TYPE

(* Data type *)
TYPE en_SYS_Objects :
(
	EO_SYS		:=0,  (* PLC *)
	EO_VPN		:=1,  (* VPN *)
	EO_DOOR		:=2,  (* Door & access control *)

	EO_CAL		:=10, (* Caldaia *)
	EO_CIR		:=11, (* Circolatore *)
	EO_CRON		:=12, (* Crono-termostato *)
	EO_VRD		:=13, (* Valvola miscelatore pannelli *)
	EO_CTL		:=14, (* Contalitri *)
	EO_CTB		:=15, (* Contabilizzatore *)
	EO_TPV		:=16, (* Temperature probes values *)
	EO_PPV		:=17, (* Pressure probes values *)
	EO_PBV		:=18, (* Over-Pressure Alarms *)
	EO_TBV		:=19, (* Over-Temperature Alarms *)
	EO_PMV		:=20, (* Under-Pressure Alarms *)
	EO_GRU		:=21, (* Gruppo termico *)
	EO_PDC		:=22, (* Pompa di calore *)
	EO_SOL		:=23, (* Pannello solare termico *)
	EO_ESOL		:=24, (* Pannello solare fotovoltaico *)
	EO_GAS		:=25, (* Contatore GAS *)
	EO_PORT		:=26, (* Misuratore di portata *)
	EO_FPV		:=27, (* Flow probes values *)
	EO_ANZ		:=28, (* Analizzatore di rete *)
	EO_SCA		:=29, (* Signal Control Alarms *)
	EO_LUX		:=30, (* Base Illumination point *)
	EO_LUXM		:=31, (* Metered Illumination point *)
	EO_PSG		:=32, (* Sensore di passaggio *)
	EO_HVAC		:=33, (* Heating, Ventilating and Air Conditioning *)
	EO_HYGRV	:=34, (* Relative Humidity sensors value *)
	EO_COOV		:=35, (* Carbon Dioxide CO2 sensors value *)
	EO_INV		:=36, (* Inverter *)
	EO_STR		:=37, (* Smart string box *)

	EO_CIRD		:=39, (* Double CIR *)
	EO_ACS		:=40, (* Hot domestic water *)
	EO_FRG		:=41, (* Frigo *)
	EO_THER		:=42, (* Thermostat *)

	EO_ZGW			:=200,  (* ZigBee - Gateway *)
	EO_ZRM			:=201,	(* ZigBee - Repeater *)
	EO_ZREL			:=202,	(* ZigBee - Actuator rele *)
	EO_ZTHL			:=203,	(* ZigBee - Temperature Sensor *)

	EO_ASGW			:=250,	(* ASi - Gateway *)
	EO_ASCBI		:=251,	(* ASi - Input Board, Ciabatta *)

	EO_LON			:=1000, (* Bus - LON *)
	EO_MODBUS		:=1001, (* Bus - MODBUS *)
	EO_MBUS			:=1002, (* Bus - M-BUS *)
	EO_MODBUS_TCP	:=1003, (* Bus - MODBUS TCP *)

	EO_GENERIC		:=9000, (* Generic dataset *)
	EO_EXPO			:=9001 (* EXPO dataset *)
);
END_TYPE

(* Data type *)
TYPE en_SYS_Status :
(
	S_UNKNOWN  := 0,
	S_STARTUP,
	S_INIT_RTC,
	S_INIT_VAR,
	S_AUTOTEST,
	S_RUNNING,
	S_SHUTDOWN,
	S_HALT
);
END_TYPE

(* Data type in LON/Enumerations *)
TYPE file_request_t :
(
	FR_NUL := -1,
	FR_OPEN_TO_SEND := 0,
	FR_OPEN_TO_RECEIVE := 1,
	FR_CLOSE_FILE := 2,
	FR_CLOSE_DELETE_FILE := 3,
	FR_DIRECTORY_LOOKUP := 4,
	FR_OPEN_TO_SEND_RA := 5,
	FR_OPEN_TO_RECEIVE_RA := 6
);
END_TYPE

(* Data type in LON/Enumerations *)
TYPE file_status_t :
(
	FS_NUL := -1,
	FS_XFER_OK := 0,
	FS_LOOKUP_OK := 1,
	FS_OPEN_FAIL := 2,
	FS_LOOKUP_ERR := 3,
	FS_XFER_UNDERWAY := 4,
	FS_IO_ERR := 5,
	FS_TIMEOUT_ERR := 6,
	FS_WINDOW_ERR := 7,
	FS_AUTH_ERR := 8,
	FS_ACCESS_UNAVAIL := 9,
	FS_SEEK_INVALID := 10,
	FS_SEEK_WAIT := 11
);
END_TYPE

(* Data type in LON/Enumerations *)
TYPE hvac_t :
(
	HVAC_NUL := -1,
	HVAC_AUTO := 0,
	HVAC_HEAT := 1,
	HVAC_MRNG_WRMUP := 2,
	HVAC_COOL := 3,
	HVAC_NIGHT_PURGE := 4,
	HVAC_PRE_COOL := 5,
	HVAC_OFF := 6,
	HVAC_TEST := 7,
	HVAC_EMERG_HEAT := 8,
	HVAC_FAN_ONLY := 9,
	HVAC_FREE_COOL := 10,
	HVAC_ICE := 11,
	HVAC_MAX_HEAT := 12,
	HVAC_ECONOMY := 13,
	HVAC_DEHUMID := 14,
	HVAC_CALIBRATE := 15,
	HVAC_EMERG_COOL := 16,
	HVAC_EMERG_STEAM := 17,
	HVAC_MAX_COOL := 18,
	HVAC_HVC_LOAD := 19,
	HVAC_NO_LOAD := 20
);
END_TYPE

(* Data type in LON/Enumerations *)
TYPE object_request_t :
(
	RQ_NUL := -1,
	RQ_NORMAL := 0,
	RQ_DISABLED := 1,
	RQ_UPDATE_STATUS := 2,
	RQ_SELF_TEST := 3,
	RQ_UPDATE_ALARM := 4,
	RQ_REPORT_MASK := 5,
	RQ_OVERRIDE := 6,
	RQ_ENABLE := 7,
	RQ_RMV_OVERRIDE := 8,
	RQ_CLEAR_STATUS := 9,
	RQ_CLEAR_ALARM := 10,
	RQ_ALARM_NOTIFY_ENABLED := 11,
	RQ_ALARM_NOTIFY_DISABLED := 12,
	RQ_MANUAL_CTRL := 13,
	RQ_REMOTE_CTRL := 14,
	RQ_PROGRAM := 15,
	RQ_CLEAR_RESET := 16,
	RQ_RESET := 17,
	RQ_CLEAR_LOG := 18,
	RQ_LOAD_PROGRAM := 19,
	RQ_RUN_PROGRAM := 20,
	RQ_HALT_PROGRAM := 21,
	RQ_RESTART_PROGRAM := 22,
	RQ_UNLOAD_PROGRAM := 23,
	RQ_STEP_PROGRAM := 24
);
END_TYPE

(* Data type in LON/Enumerations *)
TYPE priority_level_t :
(
	PR_NUL := -1,
	PR_LEVEL_0 := 0,
	PR_LEVEL_1 := 1,
	PR_LEVEL_2 := 2,
	PR_LEVEL_3 := 3,
	PR_1 := 4,
	PR_2 := 5,
	PR_3 := 6,
	PR_4 := 7,
	PR_6 := 8,
	PR_8 := 9,
	PR_10 := 10,
	PR_16 := 11
);
END_TYPE

(* Data type in Plant_Objects *)
TYPE typ_Clima : (* CURVA CLIMATICA *)
STRUCT
	InitOK:		BOOL;
	Points: 	ARRAY [0..10] OF POINT;
END_STRUCT
END_TYPE

(* Data type in Plant_Objects *)
TYPE typ_Cron_Calendar :
STRUCT
	Profile		: ARRAY[0..384] OF BYTE;
END_STRUCT
END_TYPE

(* Data type in Plant_Objects *)
TYPE typ_Cron_Jolly :
STRUCT
	Start		: DT;
	End			: DT;
	Temp		: WORD;
	Flags		: WORD; (* B0:Enabled B1..B15:Unused *)
END_STRUCT
END_TYPE

(* Data type in Plant_Objects *)
TYPE typ_Cron_Profile :
STRUCT
	Flags		: WORD;
	Setpoint	: ARRAY [0..95] OF WORD;
END_STRUCT
END_TYPE

(* Data type in Logger *)
TYPE typ_Logger :
STRUCT
	Status		: en_Logger_Status;

	SendReq		: BOOL;
	SendIdx		: DWORD;
	SendData	: ARRAY [0..MAX_SEND_TCP_CLIENT] OF BYTE;
	SendLen		: DINT;

	TData		: ARRAY [0..MAX_SEND_TCP_CLIENT] OF BYTE;
	TLen		: DINT;

	LastIdxPos	: DWORD;

	(* Temporary variables used by objects *)
	s1			: STRING(256);
	i1			: WORD;

END_STRUCT
END_TYPE

(* Data type in Plant_Objects *)
TYPE typ_MODBUS_ABB_DMTME72 :
STRUCT
	V_3P		: DWORD; (* V *)
	V_L1N		: DWORD;
	V_L2N		: DWORD;
	V_L3N		: DWORD;
	V_L1L2		: DWORD;
	V_L2L3		: DWORD;
	V_L3L1		: DWORD;
	I_3P		: DWORD; (* 10^-3 A *)
	I_L1		: DWORD;
	I_L2		: DWORD;
	I_L3		: DWORD;
	PF_3P		: DINT;	 (* 10^-3 *)
	PF_L1		: DINT;
	PF_L2		: DINT;
	PF_L3		: DINT;
	COS_3P		: DINT;  (*NO!*)
	COS_L1		: DINT;
	COS_L2		: DINT;
	COS_L3		: DINT;
	VA_3P		: DWORD; (* VA *)(*NO!*)
	VA_L1		: DWORD;
	VA_L2		: DWORD;
	VA_L3		: DWORD;
	P_3P		: DWORD; (* W *)
	P_L1		: DWORD;
	P_L2		: DWORD;
	P_L3		: DWORD;
	Q_3P		: DWORD; (* VAr *)
	Q_L1		: DWORD;
	Q_L2		: DWORD;
	Q_L3		: DWORD;

	WH_3P		: DWORD; (* 10^-1 kWh *)
	VARH_3P		: DWORD; (* 10^-1 kVArh *)
	FREQ		: DWORD; (* 10^-3 Hz *)

	I_L1_Max	: DWORD;
	I_L2_Max	: DWORD;
	I_L3_Max	: DWORD;
	P_3P_Max	: DWORD;
	Q_3P_Max	: DWORD;
	P_3P_Avg15m	: DWORD;

END_STRUCT
END_TYPE

(* Data type in Plant_Objects *)
TYPE typ_MODBUS_CIR :
STRUCT
	PumpStatus		:	WORD;
	PumpFault		:	BOOL;
	PumpBoardTemp	:	INT;	(* Electonic board temperature  [°C] *)
	PumpVoltage		:	WORD;	(* Input voltage rms [V] *)
	PumpCurrent		:	WORD;	(* Output current [E-3 A]	*)
	PumpRPM			:	WORD;	(* Round per minute [rpm] *)
	PumpPower		:	WORD;	(* Power [W] *)
	PumpOpTime		:	DWORD;	(* Pump operating time [h] *)
	PumpHead		:	WORD;	(* [E-1 m] *)
	PumpFlow		:	WORD;	(* Extimated flow [E-1 m3/h] *)
	PumpLiqTemp		:	WORD;	(* Liquid temperature [°C] *)
	PumpAlarm		:	ARRAY [0..14] OF WORD;

END_STRUCT
END_TYPE

(* Data type in Plant_Objects *)
TYPE typ_MODBUS_ELGAS_MINIELCOR :
STRUCT
	Vb			: ARRAY [0..3] OF WORD;	(* m^3 *)
	Vm			: DWORD;				(* m^3 *)
	P			: REAL;					(* bar *)
	T			: REAL;					(* °C *)
	C			: REAL;
	Vbs			: ARRAY [0..3] OF WORD;	(* m^3 *)
	Vb_d_d		: ARRAY [0..3] OF WORD;	(* m^3 *)
	Vb_d_m		: ARRAY [0..3] OF WORD;	(* m^3 *)
	Vm_d_d		: DWORD;				(* m^3 *)
	Q			: REAL;					(* m^3/h *)
	Qb			: REAL;					(* m^3/h *)

	BC_EVC		: REAL;			(* % *)
	BV_EVC		: REAL;			(* V *)
	D_Err		: WORD;			(* 0:OK, 1:FAIL *)
	Status		: DWORD;		(* Status bits *)

END_STRUCT
END_TYPE

(* Data type in Plant_Objects *)
TYPE typ_MODBUS_FRER_IQ96U2 :
STRUCT
	V_L1N		: DWORD; (* 10^-3 V *)
	V_L2N		: DWORD;
	V_L3N		: DWORD;
	V_L1L2		: DWORD;
	V_L2L3		: DWORD;
	V_L3L1		: DWORD;
	I_L1		: DWORD; (* 10^-3 I *)
	I_L2		: DWORD;
	I_L3		: DWORD;
	FREQ		: DWORD; (* 10^-3 Hz *)
	P_3P		: DWORD; (* W *)
	Q_3P		: DWORD; (* VAr *)
	PF_3P		: DINT;	 (* 10^-3 *)
	WH_3P		: DWORD; (* Wh *)
	VARH_3P		: DWORD; (* VArh *)
	MULT		: DWORD;

	WH_3P_NEG	: DWORD; (* Wh *)
	VARH_3P_NEG : DWORD; (* VArh *)
	S_3P		: DWORD; (* VA *)

	PF_L1		: DWORD; (* 10^-3 *)
	PF_L2		: DWORD; (* 10^-3 *)
	PF_L3		: DWORD; (* 10^-3 *)

	P_3P_Max	: DWORD;
	P_3P_Avg15m	: DWORD;
	I_L1_Max	: DWORD;
	I_L2_Max	: DWORD;
	I_L3_Max	: DWORD;
	I_L1_Avg15m	: DWORD;
	I_L2_Avg15m	: DWORD;
	I_L3_Avg15m	: DWORD;

END_STRUCT
END_TYPE

(* Data type in Plant_Objects *)
TYPE typ_MODBUS_VAR : (* Gestione parametri MODBUS *)
STRUCT
	SlaveAddress	: BYTE;
	FunCode			: BYTE;
	FunAddress		: WORD;
	Refresh_Time	: BYTE; (* 0:No refresh x:Refresh in seconds *)
	Refresh_Cnt		: BYTE; (* INTERNAL *)
	Variable		: POINTER TO WORD;
	Variable_Size	: BYTE;
	Variable_Mirror : WORD; (* INTERNAL [Force refresh on read variables when <>0] *)
END_STRUCT
END_TYPE

(* Data type *)
TYPE typ_SYS :
STRUCT
	Status			: en_SYS_Status;
	Warning			: BOOL;
	Alarm			: BOOL;
	AlarmStop		: BOOL;

	Time_LogString	: STRING;
	Time_Year		: WORD;
	Time_Month		: BYTE;
	Time_Day		: BYTE;

	Time_CT_DT		: DT;
	Time_CT_Day		: WORD;
	Time_CT_Quarter	: BYTE;

	LastLogs_Idx	: BYTE;
	LastLogs_Dat	: ARRAY[0..5] OF STRING;
	LastLogs_Msg	: ARRAY[0..5] OF STRING;

END_STRUCT
END_TYPE

(* Data type in Plant_Objects *)
TYPE typ_VisuStrutturaMbus :
STRUCT

	sdNodoPresente: STRING(16);
	sdEnergia: STRING(16);
	sdPotenza: STRING(16);
	sdVolume: STRING(16);
	sdFlow: STRING(16);
	sdTempIngresso: STRING(8);
	sdTempaUscita: STRING(8);
	sdTempDelta: STRING(8);

END_STRUCT
END_TYPE

(* Data type in LON/NetworkVariables *)
TYPE typSnvtAlarm : 
STRUCT
	abLocation : ARRAY[0..5] OF BYTE;
	wObjectId : WORD;
	bAlarmType : BYTE (* enum type alarm_type_t *);
	bPriorityLevel : BYTE (* enum type priority_level_t *);
	wIndexToSnvt : WORD;
	abValue : ARRAY[0..3] OF BYTE;
	wYear : WORD;
	bMonth : BYTE;
	bDay : BYTE;
	bHour : BYTE;
	bMinute : BYTE;
	bSecond : BYTE;
	wMillisecond : WORD;
	abAlarmLimit : ARRAY[0..3] OF BYTE;
	bStatusInformation : BYTE; (* bit allocation of bStatusInformation:
	bit 0: NVI update counter LSB
	bit 1: NVI update counter
	bit 2: NVI update counter
	bit 3: NVI update counter MSB
	bit 4: timeout for NVI occurs (MaxRcvTime expired)
	bit 5: reserved
	bit 6: reserved
	bit 7: force NVO update *)
	bInternalUseOnly : BYTE; (* Do not use this byte in your application! *)
END_STRUCT
END_TYPE

(* Data type in LON/NetworkVariables *)
TYPE typSnvtFilePos : 
STRUCT
	diRwPtr : DINT;
	wRwLength : WORD;
	bStatusInformation : BYTE; (* bit allocation of bStatusInformation:
	bit 0: NVI update counter LSB
	bit 1: NVI update counter
	bit 2: NVI update counter
	bit 3: NVI update counter MSB
	bit 4: timeout for NVI occurs (MaxRcvTime expired)
	bit 5: reserved
	bit 6: reserved
	bit 7: force NVO update *)
	bInternalUseOnly : BYTE; (* Do not use this byte in your application! *)
END_STRUCT
END_TYPE

(* Data type in LON/NetworkVariables *)
TYPE typSnvtFileReq : 
STRUCT
	bRequest : BYTE (* enum type file_request_t *);
	wIndex : WORD;
	wReceiveTimeout : WORD;
	abDestAddress : ARRAY[0..4] OF BYTE (* union declaration *);
	bAuthOn : BYTE;
	bPrioOn : BYTE;
	bStatusInformation : BYTE; (* bit allocation of bStatusInformation:
	bit 0: NVI update counter LSB
	bit 1: NVI update counter
	bit 2: NVI update counter
	bit 3: NVI update counter MSB
	bit 4: timeout for NVI occurs (MaxRcvTime expired)
	bit 5: reserved
	bit 6: reserved
	bit 7: force NVO update *)
	bInternalUseOnly : BYTE; (* Do not use this byte in your application! *)
END_STRUCT
END_TYPE

(* Data type in LON/NetworkVariables *)
TYPE typSnvtFileStatus : 
STRUCT
	bStatus : BYTE (* enum type file_status_t *);
	wNumberOfFiles : WORD;
	wSelectedFile : WORD;
	abAdr : ARRAY[0..21] OF BYTE (* union declaration *);
	bStatusInformation : BYTE; (* bit allocation of bStatusInformation:
	bit 0: NVI update counter LSB
	bit 1: NVI update counter
	bit 2: NVI update counter
	bit 3: NVI update counter MSB
	bit 4: timeout for NVI occurs (MaxRcvTime expired)
	bit 5: reserved
	bit 6: reserved
	bit 7: force NVO update *)
	bInternalUseOnly : BYTE; (* Do not use this byte in your application! *)
END_STRUCT
END_TYPE

(* Data type in LON/NetworkVariables *)
TYPE typSnvtHvacMode : 
STRUCT
	bSnvtHvacMode : BYTE (* enum type hvac_t *);
	bStatusInformation : BYTE; (* bit allocation of bStatusInformation:
	bit 0: NVI update counter LSB
	bit 1: NVI update counter
	bit 2: NVI update counter
	bit 3: NVI update counter MSB
	bit 4: timeout for NVI occurs (MaxRcvTime expired)
	bit 5: reserved
	bit 6: reserved
	bit 7: force NVO update *)
	bInternalUseOnly : BYTE; (* Do not use this byte in your application! *)
END_STRUCT
END_TYPE

(* Data type in LON/NetworkVariables *)
TYPE typSnvtObjRequest : 
STRUCT
	wObjectId : WORD;
	bObjectRequest : BYTE (* enum type object_request_t *);
	bStatusInformation : BYTE; (* bit allocation of bStatusInformation:
	bit 0: NVI update counter LSB
	bit 1: NVI update counter
	bit 2: NVI update counter
	bit 3: NVI update counter MSB
	bit 4: timeout for NVI occurs (MaxRcvTime expired)
	bit 5: reserved
	bit 6: reserved
	bit 7: force NVO update *)
	bInternalUseOnly : BYTE; (* Do not use this byte in your application! *)
END_STRUCT
END_TYPE

(* Data type in LON/NetworkVariables *)
TYPE typSnvtObjStatus : 
STRUCT
	wObjectId : WORD;
	bBitfieldByteOffset2 : BYTE (* bit field *);
	bBitfieldByteOffset3 : BYTE (* bit field *);
	bBitfieldByteOffset4 : BYTE (* bit field *);
	bBitfieldByteOffset5 : BYTE (* bit field *);
	bStatusInformation : BYTE; (* bit allocation of bStatusInformation:
	bit 0: NVI update counter LSB
	bit 1: NVI update counter
	bit 2: NVI update counter
	bit 3: NVI update counter MSB
	bit 4: timeout for NVI occurs (MaxRcvTime expired)
	bit 5: reserved
	bit 6: reserved
	bit 7: force NVO update *)
	bInternalUseOnly : BYTE; (* Do not use this byte in your application! *)
END_STRUCT
END_TYPE

(* Data type in LON/NetworkVariables *)
TYPE typSnvtState : 
STRUCT
	bBitfieldByteOffset0 : BYTE (* bit field *);
	bBitfieldByteOffset1 : BYTE (* bit field *);
	bStatusInformation : BYTE; (* bit allocation of bStatusInformation:
	bit 0: NVI update counter LSB
	bit 1: NVI update counter
	bit 2: NVI update counter
	bit 3: NVI update counter MSB
	bit 4: timeout for NVI occurs (MaxRcvTime expired)
	bit 5: reserved
	bit 6: reserved
	bit 7: force NVO update *)
	bInternalUseOnly : BYTE; (* Do not use this byte in your application! *)
END_STRUCT
END_TYPE

(* Data type in LON/NetworkVariables *)
TYPE typSnvtSwitch : 
STRUCT
	bValue : BYTE;
	siState : SINT;
	bStatusInformation : BYTE; (* bit allocation of bStatusInformation:
	bit 0: NVI update counter LSB
	bit 1: NVI update counter
	bit 2: NVI update counter
	bit 3: NVI update counter MSB
	bit 4: timeout for NVI occurs (MaxRcvTime expired)
	bit 5: reserved
	bit 6: reserved
	bit 7: force NVO update *)
	bInternalUseOnly : BYTE; (* Do not use this byte in your application! *)
END_STRUCT
END_TYPE

(* Data type in LON/NetworkVariables *)
TYPE typSnvtTempP :
STRUCT
	iSnvtTempP : INT;
	bStatusInformation : BYTE; (* bit allocation of bStatusInformation:
	bit 0: NVI update counter LSB
	bit 1: NVI update counter
	bit 2: NVI update counter
	bit 3: NVI update counter MSB
	bit 4: timeout for NVI occurs (MaxRcvTime expired)
	bit 5: reserved
	bit 6: reserved
	bit 7: force NVO update *)
	bInternalUseOnly : BYTE; (* Do not use this byte in your application! *)
END_STRUCT
END_TYPE

(* Data type in LON/NetworkVariables *)
TYPE typSnvtTimeStamp : 
STRUCT
	iYear : INT;
	bMonth : BYTE;
	bDay : BYTE;
	bHour : BYTE;
	bMinute : BYTE;
	bSecond : BYTE;
	bStatusInformation : BYTE; (* bit allocation of bStatusInformation:
	bit 0: NVI update counter LSB
	bit 1: NVI update counter
	bit 2: NVI update counter
	bit 3: NVI update counter MSB
	bit 4: timeout for NVI occurs (MaxRcvTime expired)
	bit 5: reserved
	bit 6: reserved
	bit 7: force NVO update *)
	bInternalUseOnly : BYTE; (* Do not use this byte in your application! *)
END_STRUCT
END_TYPE

(* POU PLC_PRG, ST *)
PROGRAM PLC_PRG
VAR
	Timer1: TON; (* Fast controls tick *)
	Timer2: TON; (* Plant control tick *)
	Timer3: TON; (* Logger timer *)

	T_CIRD01	:	INT;
	T_CIRD02	:	INT;
	T_CIRD03	:	INT;
	T_CIRD04	:	INT;
	T_CIRD05	:	INT;
	T_CIRD06	:	INT;

	SecCircuitLogic	:	BOOL;	(* Secondary circuit request: LOGICAL ON/OFF *)
	SecCircuitReal	:	BOOL;	(* Secondart circuit request: REAL ON/OFF	 *)

END_VAR
(******************************************************************************
 ****                           MAIN TASK CODE                             ****
 ******************************************************************************

	Network setup:
		IP  = 192.168.100.2 | MSK = 255.255.255.0
		GW	= 192.168.100.1 | DNS = 192.168.100.1
		SNTP = 193.204.114.232 (3600s) ==> 192.168.100.3

*)

(*==============================*)
(*===== Main status machine ====*)
(*==============================*)
Main_Stm();

(*==============================*)
(*== Running cycle operations ==*)
(*==============================*)
IF SYS.Status>S_INIT_VAR THEN

	(* Update LON output variables (needs to be here to obtain only one refresh) *)
	CAL01.Heartbeat( CLIM:=CAL01_Clima );
	CAL02.Heartbeat( CLIM:=CAL02_Clima );

	(* Execute LON process *)
	Module_1_PRG();

	(* Count water pulses *)
	CTL01(CTL_ST:=CTL01_ST, COUNT:=Ctl01_Counter);
	CTL02(CTL_ST:=CTL02_ST, COUNT:=Ctl02_Counter);

	(* ModBus *)
	MODB01();

	CIR01(ModBus:=MODB01, Pump_AL:=NOT CIR01_AL, Pump_AUTO:=NOT CIR01_AUTO, OnOff:=SecCircuitReal);
	CIR02(ModBus:=MODB01, Pump_AL:=NOT CIR02_AL, Pump_AUTO:=NOT CIR02_AUTO, Run=>CAL02.Run);

	CIRD01(ModBus:=MODB01, PumpA_AL:=NOT CIRD01_A_AL, PumpB_AL:=NOT CIRD01_B_AL, PumpA_AUTO:=NOT CIRD01_A_AUTO, PumpB_AUTO:=NOT CIRD01_B_AUTO);
	CIRD02(ModBus:=MODB01, PumpA_AL:=NOT CIRD02_A_AL, PumpB_AL:=NOT CIRD02_B_AL, PumpA_AUTO:=NOT CIRD02_A_AUTO, PumpB_AUTO:=NOT CIRD02_B_AUTO);
	CIRD03(ModBus:=MODB01, PumpA_AL:=NOT CIRD03_A_AL, PumpB_AL:=NOT CIRD03_B_AL, PumpA_AUTO:=NOT CIRD03_A_AUTO, PumpB_AUTO:=NOT CIRD03_B_AUTO);
	CIRD04(ModBus:=MODB01, PumpA_AL:=NOT CIRD04_A_AL, PumpB_AL:=NOT CIRD04_B_AL, PumpA_AUTO:=NOT CIRD04_A_AUTO, PumpB_AUTO:=NOT CIRD04_B_AUTO);
	CIRD05(ModBus:=MODB01, PumpA_AL:=NOT CIRD05_A_AL, PumpB_AL:=NOT CIRD05_B_AL, PumpA_AUTO:=NOT CIRD05_A_AUTO, PumpB_AUTO:=NOT CIRD05_B_AUTO);
	CIRD06(ModBus:=MODB01, PumpA_AL:=NOT CIRD06_A_AL, PumpB_AL:=NOT CIRD06_B_AL, PumpA_AUTO:=NOT CIRD06_A_AUTO, PumpB_AUTO:=NOT CIRD06_B_AUTO);

	(* TCP ModBus *)
	MODB02();

	ZTHL04(MODBUS:=MODB02);
	ZTHL05(MODBUS:=MODB02);
	ZTHL06(MODBUS:=MODB02);
	ZTHL07(MODBUS:=MODB02);
	ZTHL08(MODBUS:=MODB02);
	ZTHL09(MODBUS:=MODB02);
	ZTHL10(MODBUS:=MODB02);
	ZTHL11(MODBUS:=MODB02);

	(* M-Bus *)
	MBUS01();

	CTB01(MBUS:=MBUS01);

END_IF

(*==============================*)
(*== System cycle operations ===*)
(*==============================*)
(* Execute TCP processes *)
Logger_Proc();
Remote_Proc();
(* Update user led *)
USRLED_Update();
(* Execute Cron Editor commands *)
CronEd();

(* Environment temperature *)
IF NOT TPV01.ERR THEN T_AMB := S01;
ELSE T_AMB := Plant_DefaultTAmb;
END_IF


(**** SIMULATION ONLY ****)
(*...*)
END_PROGRAM
ACTION Main_Stm:
CASE Sys.Status OF

	S_STARTUP:
		Sys.Status:=S_INIT_RTC;

	S_INIT_RTC:
		(* Check RTC and update from network *)
		RTC_Update();
		(* Check time *)
		IF Sys.Time_Year>2000 THEN
			Sys.Status:=S_INIT_VAR;
		END_IF

	S_INIT_VAR:
		LogEv(EL_Wrn,EO_SYS,0,1,CONCAT('System_startup_v',WORD_TO_STRING(Plant_SW_VER)));
		Sys.Status:=S_RUNNING;

	S_RUNNING:
		Timer1(IN:=NOT Timer1.Q,PT:=T#50ms);
		IF Timer1.Q THEN
			(* Update meters *)

			(* Update system checks *)
			SYS_Proc();
		END_IF

		Timer2(IN:=NOT Timer2.Q,PT:=T#500ms);
		IF Timer2.Q THEN
			(* Read current date/time *)
			RTC_Update();

			(* Secondary circuit heat request *)
			SecCircuitLogic := CIRD01.Ctrl_Run OR CIRD02.Ctrl_Run OR CIRD03.Ctrl_Run OR CIRD04.Ctrl_Run OR CIRD05.Ctrl_Run OR CIRD06.Ctrl_Run;
			SecCircuitReal	:= CIRD01.Run OR CIRD02.Run OR CIRD03.Run OR CIRD04.Run OR CIRD05.Run OR CIRD06.Run;

			(* Boiler *)
			(*CAL01.Run:= CIR01.Run AND SYS.AlarmStop=FALSE;*)

			(* No secondary circuit heat request -->> Switch off immediatly CAL
			   Secondary circuit heat request -->> First switch on primary pump CIR01, when enabled switch on CAL *)
			CAL01.Run := SEL(SecCircuitLogic,FALSE,CIR01.Run) AND SYS.AlarmStop=FALSE;

			(* Boilers cascade *)
			CAS01(RUN_Primary:=CAL01.Run, SetTemp:=CAL01.Curve_Temp , ReadTemp:=CAL01.CFD_Temp.iSnvtTempP, OUT_Secondary=>CIR02.OnOff);


			CAL01(CLIM:=CAL01_Clima);
			CAL02(CLIM:=CAL02_Clima);

			(* Thermostats *)
			THER01(Temperature:=T_CIRD01, Run=>CIRD01.OnOff, AntifreezeForce=>CIRD01.CIR_RUN_REQ);
			THER02(Temperature:=T_CIRD02, Run=>CIRD02.OnOff, AntifreezeForce=>CIRD02.CIR_RUN_REQ);
			THER03(Temperature:=T_CIRD03, Run=>CIRD03.OnOff, AntifreezeForce=>CIRD03.CIR_RUN_REQ);
			THER04(Temperature:=T_CIRD04, Run=>CIRD04.OnOff, AntifreezeForce=>CIRD04.CIR_RUN_REQ);
			THER05(Temperature:=T_CIRD05, Run=>CIRD05.OnOff, AntifreezeForce=>CIRD05.CIR_RUN_REQ);
			THER06(Temperature:=T_CIRD06, Run=>CIRD06.OnOff, AntifreezeForce=>CIRD06.CIR_RUN_REQ);

			(* Probes *)
			TPV01(IN:=S01);
			TPV02(IN:=S02);
			TPV03(IN:=S03);

			(* Check plant status *)
			Lamp();

			(* Test toggle *)
			(*IF TEST1 THEN TEST1:=FALSE; ELSE TEST1:=TRUE; END_IF*)
		END_IF

		Timer3(IN:=NOT Timer3.Q,PT:=T#5m);
		IF Timer3.Q THEN
			(* Trig logger *)
			LogTrig();
			(* Execute temporary CSV logger *)
			(*CSV_Log();*)
		END_IF

	S_SHUTDOWN:
		(* Stop sistema *)
		Sys.Status:=S_STARTUP;

	S_HALT:
		(* Aspetta uscita manuale *)
		Sys.Status:=S_STARTUP;

ELSE
	Sys.Status:=S_STARTUP;
END_CASE;
END_ACTION

(* POU LON/Module_1/Module_1_PRG, FBD *)
PROGRAM Module_1_PRG
VAR
	(* Automatic added code, do not change! *)
	LonMaster : Module_1_LonMaster;
	SFPTnodeObject : Module_1_SFPTnodeObject;
	Virtualfunctionalblock : Module_1_Virtualfunctionalblock;

	InData_LON AT %IB0 : ARRAY[0..23] OF BYTE;
	OutData_LON AT %QB0 : ARRAY[0..23] OF BYTE;
	(***** End of automatic added code. *****)

	(* Add your code here. *)
	LonState: BOOL;
	LonReset: BOOL;

END_VAR
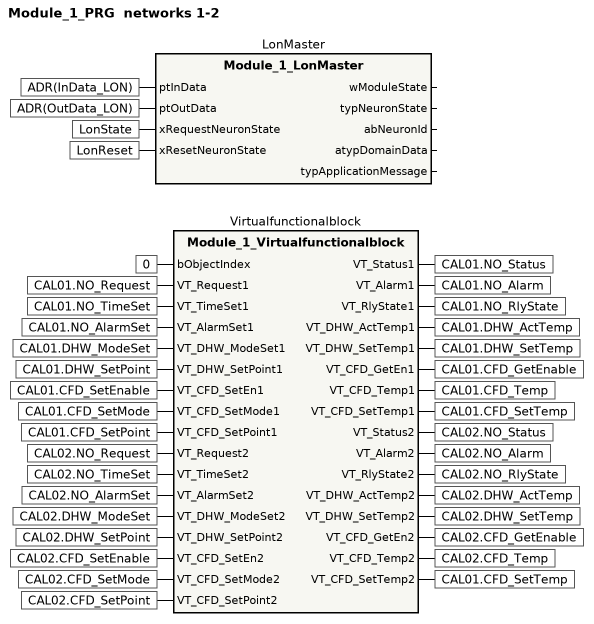
_FBD_ (* Function Block Diagram *)
NETWORK 1 (* Added by code generator *)
	LonMaster:Module_1_LonMaster(ptInData: ADR(InData_LON), ptOutData: ADR(OutData_LON), xRequestNeuronState: LonState, xResetNeuronState: LonReset)
NETWORK 2
	Virtualfunctionalblock:Module_1_Virtualfunctionalblock(bObjectIndex: 0, VT_Request1: CAL01.NO_Request, VT_TimeSet1: CAL01.NO_TimeSet, VT_AlarmSet1: CAL01.NO_AlarmSet, VT_DHW_ModeSet1: CAL01.DHW_ModeSet, VT_DHW_SetPoint1: CAL01.DHW_SetPoint, VT_CFD_SetEn1: CAL01.CFD_SetEnable, VT_CFD_SetMode1: CAL01.CFD_SetMode, VT_CFD_SetPoint1: CAL01.CFD_SetPoint, VT_Request2: CAL02.NO_Request, VT_TimeSet2: CAL02.NO_TimeSet, VT_AlarmSet2: CAL02.NO_AlarmSet, VT_DHW_ModeSet2: CAL02.DHW_ModeSet, VT_DHW_SetPoint2: CAL02.DHW_SetPoint, VT_CFD_SetEn2: CAL02.CFD_SetEnable, VT_CFD_SetMode2: CAL02.CFD_SetMode, VT_CFD_SetPoint2: CAL02.CFD_SetPoint, VT_Alarm1 => CAL01.NO_Alarm, VT_RlyState1 => CAL01.NO_RlyState, VT_DHW_ActTemp1 => CAL01.DHW_ActTemp, VT_DHW_SetTemp1 => CAL01.DHW_SetTemp, VT_CFD_GetEn1 => CAL01.CFD_GetEnable, VT_CFD_Temp1 => CAL01.CFD_Temp, VT_CFD_SetTemp1 => CAL01.CFD_SetTemp, VT_Status2 => CAL02.NO_Status, VT_Alarm2 => CAL02.NO_Alarm, VT_RlyState2 => CAL02.NO_RlyState, VT_DHW_ActTemp2 => CAL02.DHW_ActTemp, VT_DHW_SetTemp2 => CAL02.DHW_SetTemp, VT_CFD_GetEn2 => CAL02.CFD_GetEnable, VT_CFD_Temp2 => CAL02.CFD_Temp, VT_CFD_SetTemp2 => CAL01.CFD_SetTemp) => CAL01.NO_Status
_END_FBD_
(* the same logic as Structured Text *)
(* Network 1: Added by code generator *)
LonMaster(ptInData := ADR(InData_LON), ptOutData := ADR(OutData_LON), xRequestNeuronState := LonState, xResetNeuronState := LonReset);
(* Network 2 *)
Virtualfunctionalblock(bObjectIndex := 0, VT_Request1 := CAL01.NO_Request, VT_TimeSet1 := CAL01.NO_TimeSet, VT_AlarmSet1 := CAL01.NO_AlarmSet, VT_DHW_ModeSet1 := CAL01.DHW_ModeSet, VT_DHW_SetPoint1 := CAL01.DHW_SetPoint, VT_CFD_SetEn1 := CAL01.CFD_SetEnable, VT_CFD_SetMode1 := CAL01.CFD_SetMode, VT_CFD_SetPoint1 := CAL01.CFD_SetPoint, VT_Request2 := CAL02.NO_Request, VT_TimeSet2 := CAL02.NO_TimeSet, VT_AlarmSet2 := CAL02.NO_AlarmSet, VT_DHW_ModeSet2 := CAL02.DHW_ModeSet, VT_DHW_SetPoint2 := CAL02.DHW_SetPoint, VT_CFD_SetEn2 := CAL02.CFD_SetEnable, VT_CFD_SetMode2 := CAL02.CFD_SetMode, VT_CFD_SetPoint2 := CAL02.CFD_SetPoint);
CAL01.NO_Alarm := Virtualfunctionalblock.VT_Alarm1;
CAL01.NO_RlyState := Virtualfunctionalblock.VT_RlyState1;
CAL01.DHW_ActTemp := Virtualfunctionalblock.VT_DHW_ActTemp1;
CAL01.DHW_SetTemp := Virtualfunctionalblock.VT_DHW_SetTemp1;
CAL01.CFD_GetEnable := Virtualfunctionalblock.VT_CFD_GetEn1;
CAL01.CFD_Temp := Virtualfunctionalblock.VT_CFD_Temp1;
CAL01.CFD_SetTemp := Virtualfunctionalblock.VT_CFD_SetTemp1;
CAL02.NO_Status := Virtualfunctionalblock.VT_Status2;
CAL02.NO_Alarm := Virtualfunctionalblock.VT_Alarm2;
CAL02.NO_RlyState := Virtualfunctionalblock.VT_RlyState2;
CAL02.DHW_ActTemp := Virtualfunctionalblock.VT_DHW_ActTemp2;
CAL02.DHW_SetTemp := Virtualfunctionalblock.VT_DHW_SetTemp2;
CAL02.CFD_GetEnable := Virtualfunctionalblock.VT_CFD_GetEn2;
CAL02.CFD_Temp := Virtualfunctionalblock.VT_CFD_Temp2;
CAL01.CFD_SetTemp := Virtualfunctionalblock.VT_CFD_SetTemp2;
CAL01.NO_Status := Virtualfunctionalblock.VT_Status1;
END_PROGRAM

(* POU LON/Module_1/Master/Module_1_LonMaster, ST *)
FUNCTION_BLOCK Module_1_LonMaster
(******************************************)
(* Automatic generated code, do not edit! *)
(******************************************)
VAR_INPUT
	ptInData  : POINTER TO BYTE;
	ptOutData : POINTER TO BYTE;
	xRequestNeuronState : BOOL;
	xResetNeuronState : BOOL;
END_VAR
VAR_OUTPUT
	wModuleState : WORD; (* bit coded wModuleState:
	15: communication to I/O-module interrupted (error)
	14 - 08: reserved
	07: ready for Neuron initialization
	06: Neuron active
	05: user interface active
	04: internal module communication interrupted (error)
	03: CP synchronization running
	02: Neuron is configured online
	01 - 00: reserved *)

	typNeuronState : NeuronState;
	abNeuronId : ARRAY[0..5] OF BYTE;
	atypDomainData : ARRAY[0..1] OF DomainData;
	typApplicationMessage : ApplicationMessageData;
END_VAR
VAR
	bInternalCode : BYTE;
	bNvIndex : BYTE;
	wCpIndex : WORD;
	lonCom : FbLonBasicCommunication;

	xInitIsStarted : BOOL := FALSE;

	TimeoutTimer : TON;
	timeOutTime : TIME := T#1000ms;
	xStateMachineIsChecked : BOOL;
	xTimerStart : BOOL;

	iDomainTable : INT;
	xSendRequestPending : BOOL;
	trigRequest : R_TRIG;
	trigReset : R_TRIG;

	abMbxRxPrio0Buf: ARRAY [0..309] OF BYTE;
	abMbxRxPrio1Buf: ARRAY [0..517] OF BYTE;
	aMbxRxBufSize: ARRAY [0..1] OF UINT := 310, 518;
	aMbxRxBufList: ARRAY [0..1] OF POINTER TO BYTE;
	afbMbxRxFb: ARRAY [0..1] OF MBX2_RX_DEFRAG;
	astMbxRxCtx: ARRAY [0..1] OF stMbx2DefragContext;

	abMbxTxPrio0Buf: ARRAY [0..309] OF BYTE;
	abMbxTxPrio1Buf: ARRAY [0..517] OF BYTE;
	aMbxTxBufSize: ARRAY [0..1] OF UINT := 310, 518;
	aMbxTxBufList: ARRAY [0..1] OF POINTER TO BYTE;
	afbMbxTxFb: ARRAY [0..1] OF MBX2_TX_FRAG;

	astMbxTrackContext: ARRAY [0..0] OF stMbx2TrackContext;
END_VAR
VAR CONSTANT
END_VAR
aMbxRxBufList[0] := ADR(abMbxRxPrio0Buf[0]);
aMbxRxBufList[1] := ADR(abMbxRxPrio1Buf[0]);

aMbxTxBufList[0] := ADR(abMbxTxPrio0Buf[0]);
aMbxTxBufList[1] := ADR(abMbxTxPrio1Buf[0]);

mbxModule_1.Ressources.pDefragBufList := ADR(aMbxRxBufList);
mbxModule_1.Ressources.pDefragBufSizeList := ADR(aMbxRxBufSize);
mbxModule_1.Ressources.pDefragCtxPtrList := ADR(astMbxRxCtx);
mbxModule_1.Ressources.pDefragFbList := ADR(afbMbxRxFb);
mbxModule_1.Ressources.pFragBufList := ADR(aMbxTxBufList);
mbxModule_1.Ressources.pFragBufSizeList := ADR(aMbxTxBufSize);
mbxModule_1.Ressources.pFragFbList := ADR(afbMbxTxFb);

mbxModule_1.Ressources.unMaxAvailableRxPrioIndex := 1;
mbxModule_1.Ressources.unMaxAvailableTxPrioIndex := 1;

mbxModule_1.Ressources.pTrackStList := ADR(astMbxTrackContext);
mbxModule_1.Ressources.unMaxAvailableTrackIndex := 0;

mbxModule_1.Ressources.pabRxWin := ptInData + 1;
mbxModule_1.Ressources.pabTxWin := ptOutData + 1;
mbxModule_1.Ressources.bTxWinSize := 23;
mbxModule_1.Ressources.bRxWinSize := 23;

IF (mbxModule_1.bStatus.2 = TRUE) OR (mbxModule_1.bStatus.1 = TRUE) THEN
	mbxModule_1.MBX_RESET();
	xInitRunning_Module_1 := TRUE;
	xInitIsStarted := FALSE;
END_IF
mbxModule_1.MBX_CYCLE();

IF (mbxModule_1.bStatus.0 <> TRUE) THEN 
	wModuleState := 16#8000;
	RETURN;
ELSE
	wModuleState.15 := FALSE;
END_IF

xStateMachineIsChecked := FALSE;
IF xInitRunning_Module_1 = TRUE THEN
	IF xInitIsStarted = FALSE THEN
		SetParameter();
		lonCom.eInitState := INIT_SND_SGNTR_REQ;
		lonCom.CheckInitState();
		xInitIsStarted := TRUE;
		xStateMachineIsChecked := TRUE;
	END_IF
END_IF

typApplicationMessage.xMsgRcvd := FALSE;
typApplicationMessage.xRspRcvd := FALSE;
ResetNviUpdate();
WHILE (mbxModule_1.xRxPending) DO
	unLastLen_mbxModule_1 := mbxModule_1.unRxLen;
	mbxModule_1.pbRxData := ADR(InDataTelegram_Module_1);
	mbxModule_1.MBX_RETRIEVE();
	IF (mbxModule_1.nError <> MBX_OK) THEN EXIT; END_IF;
	bInternalCode := InDataTelegram_Module_1[0];

	IF (xInitRunning_Module_1 = TRUE) AND (lonCom.eInitState <> INIT_TRANSFER_CFG) THEN
		IF (FuCheckForValidInitCode(bInternalCode)) THEN
			SetParameter();
			lonCom.unLastLen := unLastLen_mbxModule_1;
			lonCom.CheckInitState();
			xInitRunning_Module_1 := NOT lonCom.xInitDone;
			xStateMachineIsChecked := TRUE;
		END_IF
	END_IF

	IF (bInternalCode = M2C_NVI_UPDT_OCCD) OR (bInternalCode = M2C_NV_VALUE_RSP) OR (bInternalCode = M2C_NVI_UPDT_TOUT) THEN
		bNvIndex := InDataTelegram_Module_1[1];
		CASE bNvIndex OF
			0, 2, 4: Module_1_PRG.SFPTnodeObject.DataReceived();
			6, 8, 10, 12, 14, 16, 18, 20, 22, 24, 26, 28, 30, 32, 34, 36: Module_1_PRG.Virtualfunctionalblock.DataReceived();

		END_CASE;
	ELSIF (bInternalCode = M2C_CP_VALUE_RSP) THEN
		wCpIndex := InDataTelegram_Module_1[1] OR (InDataTelegram_Module_1[2] * 256);
		CASE wCpIndex OF

		END_CASE;
	ELSIF (bInternalCode = M2C_LON_MSG_RCVD) OR (bInternalCode = M2C_LON_RSP_RCVD) THEN
		ApplMsgReceived();
	ELSIF (bInternalCode = M2C_STATUS_RSP) THEN
		wModuleState := (wModuleState AND 16#FF00) + InDataTelegram_Module_1[1];
	ELSIF (bInternalCode = M2C_NEURON_ID) THEN
		FuMemCopy(ADR(InDataTelegram_Module_1[1]), ADR(abNeuronId), 6);
	ELSIF (bInternalCode = M2C_DOMAIN_DATA) THEN
		DomainDataRcvd();
	ELSIF (bInternalCode = M2C_MICRO_SERVER_STATUS_RSP) THEN
		NeuronStateRcvd();
	END_IF
END_WHILE

IF (xInitRunning_Module_1 = TRUE) AND ((lonCom.xCallStateMachine = TRUE) OR (TimeoutTimer.Q = TRUE)) AND (NOT xStateMachineIsChecked) THEN
	SetParameter();
	lonCom.xTimeOut := TimeoutTimer.Q;
	lonCom.CheckInitState();
END_IF
TimeoutTimer(IN:=lonCom.xTimerStart, PT:=timeOutTime);

trigRequest(CLK := xRequestNeuronState);
trigReset(CLK := xResetNeuronState);
IF (trigRequest.Q OR trigReset.Q) THEN
	RequestNeuronState();
END_IF
END_FUNCTION_BLOCK
ACTION ApplMsgReceived:
IF (InDataTelegram_Module_1[0] = M2C_LON_MSG_RCVD) THEN
	typApplicationMessage.typService := InDataTelegram_Module_1[1] AND 16#30;
	typApplicationMessage.bSourceSubnetId := InDataTelegram_Module_1[2];
	typApplicationMessage.bSourceNodeId := InDataTelegram_Module_1[3];
	typApplicationMessage.bCorrelator := InDataTelegram_Module_1[4];
	typApplicationMessage.bCode :=  InDataTelegram_Module_1[5];
	typApplicationMessage.bDataLength := UINT_TO_BYTE(unLastLen_mbxModule_1 - 6);
	IF typApplicationMessage.bDataLength > 48 THEN typApplicationMessage.bDataLength := 48; END_IF;
	FuMemSet(ADR(typApplicationMessage.abData), 0, SIZEOF(typApplicationMessage.abData));
	IF typApplicationMessage.bDataLength > 0 THEN
		FuMemCopy(ADR(InDataTelegram_Module_1[6]), ADR(typApplicationMessage.abData), typApplicationMessage.bDataLength);
	END_IF
	typApplicationMessage.xMsgRcvd := TRUE;
ELSE
	typApplicationMessage.typService := LON_RESPONSE;
	typApplicationMessage.bSourceSubnetId := InDataTelegram_Module_1[1];
	typApplicationMessage.bSourceNodeId := InDataTelegram_Module_1[2];
	typApplicationMessage.bCorrelator := 0;
	typApplicationMessage.bCode :=  InDataTelegram_Module_1[3];
	typApplicationMessage.bDataLength := UINT_TO_BYTE(unLastLen_mbxModule_1 - 4);
	IF typApplicationMessage.bDataLength > 48 THEN typApplicationMessage.bDataLength := 48; END_IF;
	FuMemSet(ADR(typApplicationMessage.abData), 0, SIZEOF(typApplicationMessage.abData));
	IF typApplicationMessage.bDataLength > 0 THEN
		FuMemCopy(ADR(InDataTelegram_Module_1[4]), ADR(typApplicationMessage.abData), typApplicationMessage.bDataLength);
	END_IF
	typApplicationMessage.xRspRcvd := TRUE;
END_IF
END_ACTION
ACTION DomainDataRcvd:
IF (unLastLen_mbxModule_1 = 17) THEN
	iDomainTable := InDataTelegram_Module_1[1];
	IF (iDomainTable < 0) OR (iDomainTable > 1) THEN RETURN; END_IF
	FuMemCopy(ADR(InDataTelegram_Module_1[2]), ADR(atypDomainData[iDomainTable].abDomainId), 6);
	atypDomainData[iDomainTable].bSubnet := InDataTelegram_Module_1[8];
	atypDomainData[iDomainTable].xIsNonClone := InDataTelegram_Module_1[9].7;
	atypDomainData[iDomainTable].bNodeId := InDataTelegram_Module_1[9] AND 16#7F;
	atypDomainData[iDomainTable].xIsInvalid := InDataTelegram_Module_1[10].7;
	atypDomainData[iDomainTable].bDomainIdLength := InDataTelegram_Module_1[10] AND 16#7F;
	FuMemCopy(ADR(InDataTelegram_Module_1[11]), ADR(atypDomainData[iDomainTable].abAuthenticationKey), 6);
END_IF
END_ACTION
ACTION NeuronStateRcvd:
IF (unLastLen_mbxModule_1 = 16) THEN
	typNeuronState.wCrcError := InDataTelegram_Module_1[1] + InDataTelegram_Module_1[2] * 256;
	typNeuronState.wTransactionTimeouts := InDataTelegram_Module_1[3] + InDataTelegram_Module_1[4] * 256;
	typNeuronState.wReceiveTransactionBuffersFull := InDataTelegram_Module_1[5] + InDataTelegram_Module_1[6] * 256;
	typNeuronState.wLostMessages := InDataTelegram_Module_1[7] + InDataTelegram_Module_1[8] * 256;
	typNeuronState.wMissedMessages := InDataTelegram_Module_1[9] + InDataTelegram_Module_1[10] * 256;
	typNeuronState.bResetCause := InDataTelegram_Module_1[11];
	typNeuronState.bNodeState := InDataTelegram_Module_1[12];
	typNeuronState.bFirmwareVersion := InDataTelegram_Module_1[13];
	typNeuronState.bLastErrorLogged := InDataTelegram_Module_1[14];
	typNeuronState.bModelNumber := InDataTelegram_Module_1[15];
END_IF
END_ACTION
ACTION RequestNeuronState:
OutDataTelegram_Module_1[0] := C2M_MICRO_SERVER_STATUS_QRY;
OutDataTelegram_Module_1[1] := BOOL_TO_BYTE(trigReset.Q);

mbxModule_1.bTxPrio := 1;
mbxModule_1.bTxProtID := 0;
mbxModule_1.pbTxData := ADR(OutDataTelegram_Module_1);
mbxModule_1.unTxLen := 2;
mbxModule_1.MBX_SEND();

IF (mbxModule_1.nError <> MBX_OK) THEN
	RETURN;
END_IF
END_ACTION
ACTION ResetNviUpdate:
Module_1_PRG.SFPTnodeObject.ResetNviUpdate();
Module_1_PRG.Virtualfunctionalblock.ResetNviUpdate();
END_ACTION
ACTION SetParameter:
lonCom.pMbx 			:= ADR(mbxModule_1);
lonCom.pInData 			:= ADR(InDataTelegram_Module_1);
lonCom.pOutData 		:= ADR(OutDataTelegram_Module_1);
lonCom.pTimer			:= ADR(TimeoutTimer);

lonCom.pActualSignature	:= ADR(abSignature_Module_1);
lonCom.pConfigBlock := ADR(abInterface_Module_1);
lonCom.wConfigSize 		:= wConfigSize_Module_1;
END_ACTION

(* POU LON/Module_1/NV_Interface/Module_1_SFPTnodeObject, ST *)
FUNCTION_BLOCK Module_1_SFPTnodeObject
(******************************************)
(* Automatic generated code, do not edit! *)
(******************************************)
VAR_INPUT
	bObjectIndex : BYTE := 0;
	nvoStatus : typSnvtObjStatus;
	nvoFileStat : typSnvtFileStatus;

END_VAR
VAR_OUTPUT
	nviRequest : typSnvtObjRequest;
	nviFileReq : typSnvtFileReq;
	nviFilePos : typSnvtFilePos;

END_VAR
VAR
	xSetOnce : BOOL := TRUE;
	xDataInUpdated : BOOL := FALSE;
	nvoStatusLast: typSnvtObjStatus;
	nvoFileStatLast: typSnvtFileStatus;

	cmd : BYTE;
	z : INT;
	bNvRelativeIdx : BYTE;
	bNvAbsoluteIdx : BYTE;
	wCpRelativeIdx : WORD;
	wCpAbsoluteIdx : WORD;
END_VAR
VAR CONSTANT
	bNvStartIndex : BYTE := 0;
	wCpStartIndex : WORD := 65535;
	bLmoCount : BYTE := 1;
END_VAR
IF (xInitRunning_Module_1 = TRUE) AND (xSetOnce = TRUE) THEN
	xSetOnce := FALSE;
	CachePointers();
	SetUpdateFlags();
END_IF

CheckUpdateFlags();
IF (xInitRunning_Module_1 = FALSE) AND (xDataInUpdated = FALSE) THEN
	IF (mbxModule_1.bStatus.0) THEN
		SendValueRequest();
	END_IF
END_IF

IF (xInitRunning_Module_1 = FALSE) AND (mbxModule_1.bStatus.0) THEN
	xSetOnce := TRUE;
	xDataInUpdated := FALSE;
	IF ((NOT FuMemCompare(ADR(nvoStatusLast), ADR(nvoStatus), ADR(nvoStatus.bStatusInformation) - ADR(nvoStatus))) OR (nvoStatus.bStatusInformation.7 = TRUE) OR (nvoStatusLast.bInternalUseOnly.1 = TRUE)) THEN
		FuSnvtObjStatusToRaw(ADR(nvoStatus), ADR(OutDataTelegram_Module_1[2]));

		bNvAbsoluteIdx := bNvStartIndex + bObjectIndex + (1 * bLmoCount);

		IF (FuDoNvoUpdate_Module_1(ADR(nvoStatus), ADR(nvoStatusLast), ADR(nvoStatus.bInternalUseOnly), ADR(nvoStatusLast.bInternalUseOnly), ADR(nvoStatus.bStatusInformation), bNvAbsoluteIdx, 6, SIZEOF(nvoStatus)) = FALSE) THEN
			RETURN;
		END_IF
	END_IF
	IF ((NOT FuMemCompare(ADR(nvoFileStatLast), ADR(nvoFileStat), ADR(nvoFileStat.bStatusInformation) - ADR(nvoFileStat))) OR (nvoFileStat.bStatusInformation.7 = TRUE) OR (nvoFileStatLast.bInternalUseOnly.1 = TRUE)) THEN
		FuSnvtFileStatusToRaw(ADR(nvoFileStat), ADR(OutDataTelegram_Module_1[2]));

		bNvAbsoluteIdx := bNvStartIndex + bObjectIndex + (3 * bLmoCount);

		IF (FuDoNvoUpdate_Module_1(ADR(nvoFileStat), ADR(nvoFileStatLast), ADR(nvoFileStat.bInternalUseOnly), ADR(nvoFileStatLast.bInternalUseOnly), ADR(nvoFileStat.bStatusInformation), bNvAbsoluteIdx, 27, SIZEOF(nvoFileStat)) = FALSE) THEN
			RETURN;
		END_IF
	END_IF

END_IF
END_FUNCTION_BLOCK
ACTION CachePointers:
;
END_ACTION
ACTION CheckUpdateFlags:
xDataInUpdated := (NOT nviRequest.bInternalUseOnly.0) AND (NOT nviFileReq.bInternalUseOnly.0) AND (NOT nviFilePos.bInternalUseOnly.0) AND TRUE;
END_ACTION
ACTION DataReceived:
cmd := InDataTelegram_Module_1[0];
IF (cmd = M2C_NVI_UPDT_OCCD) OR (cmd = M2C_NV_VALUE_RSP) OR (cmd = M2C_NVI_UPDT_TOUT) THEN
	bNvRelativeIdx := (InDataTelegram_Module_1[1] - bNvStartIndex - bObjectIndex) / bLmoCount;
	CASE bNvRelativeIdx OF
	0:
		IF (cmd = M2C_NVI_UPDT_OCCD) OR (cmd = M2C_NV_VALUE_RSP) THEN
			IF (unLastLen_mbxModule_1 = (2 + 3)) THEN
				FuRawToSnvtObjRequest(ADR(InDataTelegram_Module_1[2]), ADR(nviRequest));
				nviRequest.bInternalUseOnly.0 := FALSE;
				nviRequest.bStatusInformation := FuInkrementNviStatus(nviRequest.bStatusInformation);
			ELSIF (unLastLen_mbxModule_1 = 2) THEN
				nviRequest.bStatusInformation := FuInkrementNviStatus(nviRequest.bStatusInformation);
			END_IF
		ELSIF (cmd = M2C_NVI_UPDT_TOUT) THEN
			IF (unLastLen_mbxModule_1 = 3) THEN
				nviRequest.bStatusInformation.4 := BYTE_TO_BOOL(InDataTelegram_Module_1[2]);
			END_IF
		END_IF
	2:
		IF (cmd = M2C_NVI_UPDT_OCCD) OR (cmd = M2C_NV_VALUE_RSP) THEN
			IF (unLastLen_mbxModule_1 = (2 + 12)) THEN
				FuRawToSnvtFileReq(ADR(InDataTelegram_Module_1[2]), ADR(nviFileReq));
				nviFileReq.bInternalUseOnly.0 := FALSE;
				nviFileReq.bStatusInformation := FuInkrementNviStatus(nviFileReq.bStatusInformation);
			ELSIF (unLastLen_mbxModule_1 = 2) THEN
				nviFileReq.bStatusInformation := FuInkrementNviStatus(nviFileReq.bStatusInformation);
			END_IF
		ELSIF (cmd = M2C_NVI_UPDT_TOUT) THEN
			IF (unLastLen_mbxModule_1 = 3) THEN
				nviFileReq.bStatusInformation.4 := BYTE_TO_BOOL(InDataTelegram_Module_1[2]);
			END_IF
		END_IF
	4:
		IF (cmd = M2C_NVI_UPDT_OCCD) OR (cmd = M2C_NV_VALUE_RSP) THEN
			IF (unLastLen_mbxModule_1 = (2 + 6)) THEN
				FuRawToSnvtFilePos(ADR(InDataTelegram_Module_1[2]), ADR(nviFilePos));
				nviFilePos.bInternalUseOnly.0 := FALSE;
				nviFilePos.bStatusInformation := FuInkrementNviStatus(nviFilePos.bStatusInformation);
			ELSIF (unLastLen_mbxModule_1 = 2) THEN
				nviFilePos.bStatusInformation := FuInkrementNviStatus(nviFilePos.bStatusInformation);
			END_IF
		ELSIF (cmd = M2C_NVI_UPDT_TOUT) THEN
			IF (unLastLen_mbxModule_1 = 3) THEN
				nviFilePos.bStatusInformation.4 := BYTE_TO_BOOL(InDataTelegram_Module_1[2]);
			END_IF
		END_IF

	END_CASE
ELSIF (cmd = M2C_CP_VALUE_RSP) THEN
	wCpRelativeIdx := ((InDataTelegram_Module_1[1] + InDataTelegram_Module_1[2] * 256) - wCpStartIndex - bObjectIndex) / bLmoCount;
	CASE wCpRelativeIdx OF

	END_CASE
END_IF
END_ACTION
ACTION ResetNviUpdate:
nviRequest.bStatusInformation := nviRequest.bStatusInformation AND 16#F8;
nviFileReq.bStatusInformation := nviFileReq.bStatusInformation AND 16#F8;
nviFilePos.bStatusInformation := nviFilePos.bStatusInformation AND 16#F8;
;
END_ACTION
ACTION SendValueRequest:
IF (FuSendNviValueReq_Module_1(ADR(nviRequest.bInternalUseOnly), bNvStartIndex + bObjectIndex + (0 * bLmoCount)) = FALSE) THEN
	RETURN;
END_IF

IF (FuSendNviValueReq_Module_1(ADR(nviFileReq.bInternalUseOnly), bNvStartIndex + bObjectIndex + (2 * bLmoCount)) = FALSE) THEN
	RETURN;
END_IF

IF (FuSendNviValueReq_Module_1(ADR(nviFilePos.bInternalUseOnly), bNvStartIndex + bObjectIndex + (4 * bLmoCount)) = FALSE) THEN
	RETURN;
END_IF

;
END_ACTION
ACTION SetUpdateFlags:
nviRequest.bInternaluseOnly.0 := TRUE;
nvoStatusLast.bInternaluseOnly.1 := TRUE;
nvoStatusLast.bInternaluseOnly.7 := FALSE;
nviFileReq.bInternaluseOnly.0 := TRUE;
nvoFileStatLast.bInternaluseOnly.1 := TRUE;
nvoFileStatLast.bInternaluseOnly.7 := FALSE;
nviFilePos.bInternaluseOnly.0 := TRUE;
;
END_ACTION

(* POU LON/Shared/Internal/FuSnvtObjStatusToRaw, ST *)
FUNCTION FuSnvtObjStatusToRaw : BOOL
(******************************************)
(* Automatic generated code, do not edit! *)
(******************************************)
VAR_INPUT
	NvDataIn :  POINTER TO typSnvtObjStatus;
	DataOut : POINTER TO ARRAY[0..5] OF BYTE;
END_VAR
VAR
END_VAR
DataOut^[0] := WORD_TO_BYTE(SHR(NvDataIn^.wObjectId, 8));
DataOut^[1] := WORD_TO_BYTE(NvDataIn^.wObjectId);

DataOut^[2] := NvDataIn^.bBitfieldByteOffset2;

DataOut^[3] := NvDataIn^.bBitfieldByteOffset3;

DataOut^[4] := NvDataIn^.bBitfieldByteOffset4;

DataOut^[5] := NvDataIn^.bBitfieldByteOffset5;

FuSnvtObjStatusToRaw := TRUE;
END_FUNCTION

(* POU LON/Module_1/Internal/FuDoNvoUpdate_Module_1, ST *)
FUNCTION FuDoNvoUpdate_Module_1 : BOOL
(******************************************)
(* Automatic generated code, do not edit! *)
(******************************************)
VAR_INPUT
	ptNvo : POINTER TO BYTE;
	ptNvoLast : POINTER TO BYTE;
	ptNvoInternalUse : POINTER TO BYTE;
	ptNvoLastInternalUse : POINTER TO BYTE;
	ptNvoStatusInformation : POINTER TO BYTE;
	bNvoIndex : BYTE;
	uiNvoLength : UINT;
	uiNvoVariableLength : UINT;
END_VAR
IF (ptNvoLastInternalUse^.1 = TRUE) AND (ptNvoStatusInformation^.7 = FALSE) THEN
	OutDataTelegram_Module_1[0] := C2M_NV_VALUE;
ELSE
	OutDataTelegram_Module_1[0] := C2M_NVO_PROPAGATE;
END_IF
OutDataTelegram_Module_1[1] := bNvoIndex;

mbxModule_1.bTxPrio := BOOL_TO_BYTE(ptNvoLastInternalUse^.7);
mbxModule_1.bTxProtID := 0;
mbxModule_1.pbTxData := ADR(OutDataTelegram_Module_1);
mbxModule_1.unTxLen := 2 + uiNvoLength;
mbxModule_1.MBX_SEND();

IF (mbxModule_1.nError <> MBX_OK) THEN
	FuDoNvoUpdate_Module_1 := FALSE;
	RETURN;
END_IF

ptNvoLastInternalUse^.1 := FALSE;
ptNvoInternalUse^ := ptNvoLastInternalUse^;
FuMemCopy(ptNvo, ptNvoLast, uiNvoVariableLength);

FuDoNvoUpdate_Module_1 := TRUE;
END_FUNCTION

(* POU LON/Shared/Internal/FuSnvtFileStatusToRaw, ST *)
FUNCTION FuSnvtFileStatusToRaw : BOOL
(******************************************)
(* Automatic generated code, do not edit! *)
(******************************************)
VAR_INPUT
	NvDataIn :  POINTER TO typSnvtFileStatus;
	DataOut : POINTER TO ARRAY[0..26] OF BYTE;
END_VAR
VAR
END_VAR
DataOut^[0] := NvDataIn^.bStatus;

DataOut^[1] := WORD_TO_BYTE(SHR(NvDataIn^.wNumberOfFiles, 8));
DataOut^[2] := WORD_TO_BYTE(NvDataIn^.wNumberOfFiles);

DataOut^[3] := WORD_TO_BYTE(SHR(NvDataIn^.wSelectedFile, 8));
DataOut^[4] := WORD_TO_BYTE(NvDataIn^.wSelectedFile);

DataOut^[5] := NvDataIn^.abAdr[0];
DataOut^[6] := NvDataIn^.abAdr[1];
DataOut^[7] := NvDataIn^.abAdr[2];
DataOut^[8] := NvDataIn^.abAdr[3];
DataOut^[9] := NvDataIn^.abAdr[4];
DataOut^[10] := NvDataIn^.abAdr[5];
DataOut^[11] := NvDataIn^.abAdr[6];
DataOut^[12] := NvDataIn^.abAdr[7];
DataOut^[13] := NvDataIn^.abAdr[8];
DataOut^[14] := NvDataIn^.abAdr[9];
DataOut^[15] := NvDataIn^.abAdr[10];
DataOut^[16] := NvDataIn^.abAdr[11];
DataOut^[17] := NvDataIn^.abAdr[12];
DataOut^[18] := NvDataIn^.abAdr[13];
DataOut^[19] := NvDataIn^.abAdr[14];
DataOut^[20] := NvDataIn^.abAdr[15];
DataOut^[21] := NvDataIn^.abAdr[16];
DataOut^[22] := NvDataIn^.abAdr[17];
DataOut^[23] := NvDataIn^.abAdr[18];
DataOut^[24] := NvDataIn^.abAdr[19];
DataOut^[25] := NvDataIn^.abAdr[20];
DataOut^[26] := NvDataIn^.abAdr[21];

FuSnvtFileStatusToRaw := TRUE;
END_FUNCTION

(* POU LON/Module_1/Internal/FuSendNviValueReq_Module_1, ST *)
FUNCTION FuSendNviValueReq_Module_1 : BOOL
(******************************************)
(* Automatic generated code, do not edit! *)
(******************************************)
VAR_INPUT
	ptInternalUseOnly : POINTER TO BYTE;
	bNvIndex : BYTE;
END_VAR
IF ptInternalUseOnly^.0 = TRUE THEN
	OutDataTelegram_Module_1[0] := C2M_NV_VALUE_QRY;
	OutDataTelegram_Module_1[1] := bNvIndex;

	mbxModule_1.bTxPrio := 1;
	mbxModule_1.bTxProtID := 0;
	mbxModule_1.pbTxData := ADR(OutDataTelegram_Module_1);
	mbxModule_1.unTxLen := 2;
	mbxModule_1.MBX_SEND();

	IF (mbxModule_1.nError <> MBX_OK) THEN
		FuSendNviValueReq_Module_1 := FALSE;
		RETURN;
	END_IF
	ptInternalUseOnly^.0 := FALSE;
END_IF

FuSendNviValueReq_Module_1 := TRUE;
END_FUNCTION

(* POU LON/Module_1/NV_Interface/Module_1_Virtualfunctionalblock, ST *)
FUNCTION_BLOCK Module_1_Virtualfunctionalblock
(******************************************)
(* Automatic generated code, do not edit! *)
(******************************************)
VAR_INPUT
	bObjectIndex : BYTE := 0;
	VT_Request1 : typSnvtObjRequest;
	VT_TimeSet1 : typSnvtTimeStamp;
	VT_AlarmSet1 : typSnvtAlarm;
	VT_DHW_ModeSet1 : typSnvtHvacMode;
	VT_DHW_SetPoint1 : typSnvtTempP;
	VT_CFD_SetEn1 : typSnvtSwitch;
	VT_CFD_SetMode1 : typSnvtHvacMode;
	VT_CFD_SetPoint1 : typSnvtTempP;
	VT_Request2 : typSnvtObjRequest;
	VT_TimeSet2 : typSnvtTimeStamp;
	VT_AlarmSet2 : typSnvtAlarm;
	VT_DHW_ModeSet2 : typSnvtHvacMode;
	VT_DHW_SetPoint2 : typSnvtTempP;
	VT_CFD_SetEn2 : typSnvtSwitch;
	VT_CFD_SetMode2 : typSnvtHvacMode;
	VT_CFD_SetPoint2 : typSnvtTempP;

END_VAR
VAR_OUTPUT
	VT_Status1 : typSnvtObjStatus;
	VT_Alarm1 : typSnvtAlarm;
	VT_RlyState1 : typSnvtState;
	VT_DHW_ActTemp1 : typSnvtTempP;
	VT_DHW_SetTemp1 : typSnvtTempP;
	VT_CFD_GetEn1 : typSnvtSwitch;
	VT_CFD_Temp1 : typSnvtTempP;
	VT_CFD_SetTemp1 : typSnvtTempP;
	VT_Status2 : typSnvtObjStatus;
	VT_Alarm2 : typSnvtAlarm;
	VT_RlyState2 : typSnvtState;
	VT_DHW_ActTemp2 : typSnvtTempP;
	VT_DHW_SetTemp2 : typSnvtTempP;
	VT_CFD_GetEn2 : typSnvtSwitch;
	VT_CFD_Temp2 : typSnvtTempP;
	VT_CFD_SetTemp2 : typSnvtTempP;

END_VAR
VAR
	xSetOnce : BOOL := TRUE;
	xDataInUpdated : BOOL := FALSE;
	paNviSnvtObjStatus : ARRAY[0..1] OF POINTER TO typSnvtObjStatus;
	aNviSnvtObjStatusIndex : ARRAY[0..1] OF BYTE := 1,17;
	paNviSnvtAlarm : ARRAY[0..1] OF POINTER TO typSnvtAlarm;
	aNviSnvtAlarmIndex : ARRAY[0..1] OF BYTE := 3,19;
	paNviSnvtState : ARRAY[0..1] OF POINTER TO typSnvtState;
	aNviSnvtStateIndex : ARRAY[0..1] OF BYTE := 5,21;
	paNviSnvtTempP : ARRAY[0..7] OF POINTER TO typSnvtTempP;
	aNviSnvtTempPIndex : ARRAY[0..7] OF BYTE := 7,9,13,15,23,25,29,31;
	paNviSnvtSwitch : ARRAY[0..1] OF POINTER TO typSnvtSwitch;
	aNviSnvtSwitchIndex : ARRAY[0..1] OF BYTE := 11,27;
	paNvoSnvtObjRequest : ARRAY[0..1] OF POINTER TO typSnvtObjRequest;
	aNvoSnvtObjRequestIndex : ARRAY[0..1] OF BYTE := 0,16;
	aNvoSnvtObjRequestLast : ARRAY[0..1] OF typSnvtObjRequest;
	aNvoSnvtObjRequestPriority : ARRAY[0..0] OF BYTE := 16#00;
	paNvoSnvtTimeStamp : ARRAY[0..1] OF POINTER TO typSnvtTimeStamp;
	aNvoSnvtTimeStampIndex : ARRAY[0..1] OF BYTE := 2,18;
	aNvoSnvtTimeStampLast : ARRAY[0..1] OF typSnvtTimeStamp;
	aNvoSnvtTimeStampPriority : ARRAY[0..0] OF BYTE := 16#00;
	paNvoSnvtAlarm : ARRAY[0..1] OF POINTER TO typSnvtAlarm;
	aNvoSnvtAlarmIndex : ARRAY[0..1] OF BYTE := 4,20;
	aNvoSnvtAlarmLast : ARRAY[0..1] OF typSnvtAlarm;
	aNvoSnvtAlarmPriority : ARRAY[0..0] OF BYTE := 16#00;
	paNvoSnvtHvacMode : ARRAY[0..3] OF POINTER TO typSnvtHvacMode;
	aNvoSnvtHvacModeIndex : ARRAY[0..3] OF BYTE := 6,12,22,28;
	aNvoSnvtHvacModeLast : ARRAY[0..3] OF typSnvtHvacMode;
	aNvoSnvtHvacModePriority : ARRAY[0..0] OF BYTE := 16#00;
	paNvoSnvtTempP : ARRAY[0..3] OF POINTER TO typSnvtTempP;
	aNvoSnvtTempPIndex : ARRAY[0..3] OF BYTE := 8,14,24,30;
	aNvoSnvtTempPLast : ARRAY[0..3] OF typSnvtTempP;
	aNvoSnvtTempPPriority : ARRAY[0..0] OF BYTE := 16#00;
	paNvoSnvtSwitch : ARRAY[0..1] OF POINTER TO typSnvtSwitch;
	aNvoSnvtSwitchIndex : ARRAY[0..1] OF BYTE := 10,26;
	aNvoSnvtSwitchLast : ARRAY[0..1] OF typSnvtSwitch;
	aNvoSnvtSwitchPriority : ARRAY[0..0] OF BYTE := 16#00;

	cmd : BYTE;
	z : INT;
	bNvRelativeIdx : BYTE;
	bNvAbsoluteIdx : BYTE;
	wCpRelativeIdx : WORD;
	wCpAbsoluteIdx : WORD;
END_VAR
VAR CONSTANT
	bNvStartIndex : BYTE := 5;
	wCpStartIndex : WORD := 65535;
	bLmoCount : BYTE := 1;
END_VAR
IF (xInitRunning_Module_1 = TRUE) AND (xSetOnce = TRUE) THEN
	xSetOnce := FALSE;
	CachePointers();
	SetUpdateFlags();
END_IF

CheckUpdateFlags();
IF (xInitRunning_Module_1 = FALSE) AND (xDataInUpdated = FALSE) THEN
	IF (mbxModule_1.bStatus.0) THEN
		SendValueRequest();
	END_IF
END_IF

IF (xInitRunning_Module_1 = FALSE) AND (mbxModule_1.bStatus.0) THEN
	xSetOnce := TRUE;
	xDataInUpdated := FALSE;
	FOR z := 0 TO 1 DO
		IF ((NOT FuMemCompare(ADR(aNvoSnvtObjRequestLast[z]), paNvoSnvtObjRequest[z], ADR(paNvoSnvtObjRequest[z]^.bStatusInformation) - paNvoSnvtObjRequest[z])) OR (paNvoSnvtObjRequest[z]^.bStatusInformation.7 = TRUE) OR (aNvoSnvtObjRequestLast[z].bInternalUseOnly.1 = TRUE)) THEN
			FuSnvtObjRequestToRaw(paNvoSnvtObjRequest[z], ADR(OutDataTelegram_Module_1[2]));

			bNvAbsoluteIdx := bNvStartIndex + bObjectIndex + (aNvoSnvtObjRequestIndex[z] * bLmoCount);

			IF (FuDoNvoUpdate_Module_1(paNvoSnvtObjRequest[z], ADR(aNvoSnvtObjRequestLast[z]), ADR(paNvoSnvtObjRequest[z]^.bInternalUseOnly), ADR(aNvoSnvtObjRequestLast[z].bInternalUseOnly), ADR(paNvoSnvtObjRequest[z]^.bStatusInformation), bNvAbsoluteIdx, 3, SIZEOF(aNvoSnvtObjRequestLast[z])) = FALSE) THEN
				RETURN;
			END_IF
		END_IF
	END_FOR
	FOR z := 0 TO 1 DO
		IF ((NOT FuMemCompare(ADR(aNvoSnvtTimeStampLast[z]), paNvoSnvtTimeStamp[z], ADR(paNvoSnvtTimeStamp[z]^.bStatusInformation) - paNvoSnvtTimeStamp[z])) OR (paNvoSnvtTimeStamp[z]^.bStatusInformation.7 = TRUE) OR (aNvoSnvtTimeStampLast[z].bInternalUseOnly.1 = TRUE)) THEN
			FuSnvtTimeStampToRaw(paNvoSnvtTimeStamp[z], ADR(OutDataTelegram_Module_1[2]));

			bNvAbsoluteIdx := bNvStartIndex + bObjectIndex + (aNvoSnvtTimeStampIndex[z] * bLmoCount);

			IF (FuDoNvoUpdate_Module_1(paNvoSnvtTimeStamp[z], ADR(aNvoSnvtTimeStampLast[z]), ADR(paNvoSnvtTimeStamp[z]^.bInternalUseOnly), ADR(aNvoSnvtTimeStampLast[z].bInternalUseOnly), ADR(paNvoSnvtTimeStamp[z]^.bStatusInformation), bNvAbsoluteIdx, 7, SIZEOF(aNvoSnvtTimeStampLast[z])) = FALSE) THEN
				RETURN;
			END_IF
		END_IF
	END_FOR
	FOR z := 0 TO 1 DO
		IF ((NOT FuMemCompare(ADR(aNvoSnvtAlarmLast[z]), paNvoSnvtAlarm[z], ADR(paNvoSnvtAlarm[z]^.bStatusInformation) - paNvoSnvtAlarm[z])) OR (paNvoSnvtAlarm[z]^.bStatusInformation.7 = TRUE) OR (aNvoSnvtAlarmLast[z].bInternalUseOnly.1 = TRUE)) THEN
			FuSnvtAlarmToRaw(paNvoSnvtAlarm[z], ADR(OutDataTelegram_Module_1[2]));

			bNvAbsoluteIdx := bNvStartIndex + bObjectIndex + (aNvoSnvtAlarmIndex[z] * bLmoCount);

			IF (FuDoNvoUpdate_Module_1(paNvoSnvtAlarm[z], ADR(aNvoSnvtAlarmLast[z]), ADR(paNvoSnvtAlarm[z]^.bInternalUseOnly), ADR(aNvoSnvtAlarmLast[z].bInternalUseOnly), ADR(paNvoSnvtAlarm[z]^.bStatusInformation), bNvAbsoluteIdx, 29, SIZEOF(aNvoSnvtAlarmLast[z])) = FALSE) THEN
				RETURN;
			END_IF
		END_IF
	END_FOR
	FOR z := 0 TO 3 DO
		IF ((NOT FuMemCompare(ADR(aNvoSnvtHvacModeLast[z]), paNvoSnvtHvacMode[z], ADR(paNvoSnvtHvacMode[z]^.bStatusInformation) - paNvoSnvtHvacMode[z])) OR (paNvoSnvtHvacMode[z]^.bStatusInformation.7 = TRUE) OR (aNvoSnvtHvacModeLast[z].bInternalUseOnly.1 = TRUE)) THEN
			FuSnvtHvacModeToRaw(paNvoSnvtHvacMode[z], ADR(OutDataTelegram_Module_1[2]));

			bNvAbsoluteIdx := bNvStartIndex + bObjectIndex + (aNvoSnvtHvacModeIndex[z] * bLmoCount);

			IF (FuDoNvoUpdate_Module_1(paNvoSnvtHvacMode[z], ADR(aNvoSnvtHvacModeLast[z]), ADR(paNvoSnvtHvacMode[z]^.bInternalUseOnly), ADR(aNvoSnvtHvacModeLast[z].bInternalUseOnly), ADR(paNvoSnvtHvacMode[z]^.bStatusInformation), bNvAbsoluteIdx, 1, SIZEOF(aNvoSnvtHvacModeLast[z])) = FALSE) THEN
				RETURN;
			END_IF
		END_IF
	END_FOR
	FOR z := 0 TO 3 DO
		IF ((NOT FuMemCompare(ADR(aNvoSnvtTempPLast[z]), paNvoSnvtTempP[z], ADR(paNvoSnvtTempP[z]^.bStatusInformation) - paNvoSnvtTempP[z])) OR (paNvoSnvtTempP[z]^.bStatusInformation.7 = TRUE) OR (aNvoSnvtTempPLast[z].bInternalUseOnly.1 = TRUE)) THEN
			FuSnvtTempPToRaw(paNvoSnvtTempP[z], ADR(OutDataTelegram_Module_1[2]));

			bNvAbsoluteIdx := bNvStartIndex + bObjectIndex + (aNvoSnvtTempPIndex[z] * bLmoCount);

			IF (FuDoNvoUpdate_Module_1(paNvoSnvtTempP[z], ADR(aNvoSnvtTempPLast[z]), ADR(paNvoSnvtTempP[z]^.bInternalUseOnly), ADR(aNvoSnvtTempPLast[z].bInternalUseOnly), ADR(paNvoSnvtTempP[z]^.bStatusInformation), bNvAbsoluteIdx, 2, SIZEOF(aNvoSnvtTempPLast[z])) = FALSE) THEN
				RETURN;
			END_IF
		END_IF
	END_FOR
	FOR z := 0 TO 1 DO
		IF ((NOT FuMemCompare(ADR(aNvoSnvtSwitchLast[z]), paNvoSnvtSwitch[z], ADR(paNvoSnvtSwitch[z]^.bStatusInformation) - paNvoSnvtSwitch[z])) OR (paNvoSnvtSwitch[z]^.bStatusInformation.7 = TRUE) OR (aNvoSnvtSwitchLast[z].bInternalUseOnly.1 = TRUE)) THEN
			FuSnvtSwitchToRaw(paNvoSnvtSwitch[z], ADR(OutDataTelegram_Module_1[2]));

			bNvAbsoluteIdx := bNvStartIndex + bObjectIndex + (aNvoSnvtSwitchIndex[z] * bLmoCount);

			IF (FuDoNvoUpdate_Module_1(paNvoSnvtSwitch[z], ADR(aNvoSnvtSwitchLast[z]), ADR(paNvoSnvtSwitch[z]^.bInternalUseOnly), ADR(aNvoSnvtSwitchLast[z].bInternalUseOnly), ADR(paNvoSnvtSwitch[z]^.bStatusInformation), bNvAbsoluteIdx, 2, SIZEOF(aNvoSnvtSwitchLast[z])) = FALSE) THEN
				RETURN;
			END_IF
		END_IF
	END_FOR

END_IF
END_FUNCTION_BLOCK
ACTION CachePointers:
paNviSnvtObjStatus[0] := ADR(VT_Status1);
paNviSnvtObjStatus[1] := ADR(VT_Status2);
paNviSnvtAlarm[0] := ADR(VT_Alarm1);
paNviSnvtAlarm[1] := ADR(VT_Alarm2);
paNviSnvtState[0] := ADR(VT_RlyState1);
paNviSnvtState[1] := ADR(VT_RlyState2);
paNviSnvtTempP[0] := ADR(VT_DHW_ActTemp1);
paNviSnvtTempP[1] := ADR(VT_DHW_SetTemp1);
paNviSnvtTempP[2] := ADR(VT_CFD_Temp1);
paNviSnvtTempP[3] := ADR(VT_CFD_SetTemp1);
paNviSnvtTempP[4] := ADR(VT_DHW_ActTemp2);
paNviSnvtTempP[5] := ADR(VT_DHW_SetTemp2);
paNviSnvtTempP[6] := ADR(VT_CFD_Temp2);
paNviSnvtTempP[7] := ADR(VT_CFD_SetTemp2);
paNviSnvtSwitch[0] := ADR(VT_CFD_GetEn1);
paNviSnvtSwitch[1] := ADR(VT_CFD_GetEn2);
paNvoSnvtObjRequest[0] := ADR(VT_Request1);
paNvoSnvtObjRequest[1] := ADR(VT_Request2);
paNvoSnvtTimeStamp[0] := ADR(VT_TimeSet1);
paNvoSnvtTimeStamp[1] := ADR(VT_TimeSet2);
paNvoSnvtAlarm[0] := ADR(VT_AlarmSet1);
paNvoSnvtAlarm[1] := ADR(VT_AlarmSet2);
paNvoSnvtHvacMode[0] := ADR(VT_DHW_ModeSet1);
paNvoSnvtHvacMode[1] := ADR(VT_CFD_SetMode1);
paNvoSnvtHvacMode[2] := ADR(VT_DHW_ModeSet2);
paNvoSnvtHvacMode[3] := ADR(VT_CFD_SetMode2);
paNvoSnvtTempP[0] := ADR(VT_DHW_SetPoint1);
paNvoSnvtTempP[1] := ADR(VT_CFD_SetPoint1);
paNvoSnvtTempP[2] := ADR(VT_DHW_SetPoint2);
paNvoSnvtTempP[3] := ADR(VT_CFD_SetPoint2);
paNvoSnvtSwitch[0] := ADR(VT_CFD_SetEn1);
paNvoSnvtSwitch[1] := ADR(VT_CFD_SetEn2);
;
END_ACTION
ACTION CheckUpdateFlags:
xDataInUpdated := TRUE;
FOR z := 0 TO 1 DO
	xDataInUpdated := xDataInUpdated AND (NOT paNviSnvtObjStatus[z]^.bInternalUseOnly.0);
END_FOR
FOR z := 0 TO 1 DO
	xDataInUpdated := xDataInUpdated AND (NOT paNviSnvtAlarm[z]^.bInternalUseOnly.0);
END_FOR
FOR z := 0 TO 1 DO
	xDataInUpdated := xDataInUpdated AND (NOT paNviSnvtState[z]^.bInternalUseOnly.0);
END_FOR
FOR z := 0 TO 7 DO
	xDataInUpdated := xDataInUpdated AND (NOT paNviSnvtTempP[z]^.bInternalUseOnly.0);
END_FOR
FOR z := 0 TO 1 DO
	xDataInUpdated := xDataInUpdated AND (NOT paNviSnvtSwitch[z]^.bInternalUseOnly.0);
END_FOR
END_ACTION
ACTION DataReceived:
cmd := InDataTelegram_Module_1[0];
IF (cmd = M2C_NVI_UPDT_OCCD) OR (cmd = M2C_NV_VALUE_RSP) OR (cmd = M2C_NVI_UPDT_TOUT) THEN
	bNvRelativeIdx := (InDataTelegram_Module_1[1] - bNvStartIndex - bObjectIndex) / bLmoCount;
	CASE bNvRelativeIdx OF
	1, 17:
		IF (cmd = M2C_NVI_UPDT_OCCD) OR (cmd = M2C_NV_VALUE_RSP) THEN
			IF (unLastLen_mbxModule_1 = (2 + 6)) THEN
				FOR z := 0 TO 1 DO
					IF aNviSnvtObjStatusIndex[z] = bNvRelativeIdx THEN
						FuRawToSnvtObjStatus(ADR(InDataTelegram_Module_1[2]), paNviSnvtObjStatus[z]);
						paNviSnvtObjStatus[z]^.bInternalUseOnly.0 := FALSE;
						paNviSnvtObjStatus[z]^.bStatusInformation := FuInkrementNviStatus(paNviSnvtObjStatus[z]^.bStatusInformation);
						EXIT;
					END_IF
				END_FOR
			ELSIF (unLastLen_mbxModule_1 = 2) THEN
				FOR z := 0 TO 1 DO
					IF aNviSnvtObjStatusIndex[z] = bNvRelativeIdx THEN
						paNviSnvtObjStatus[z]^.bStatusInformation := FuInkrementNviStatus(paNviSnvtObjStatus[z]^.bStatusInformation);
						EXIT;
					END_IF
				END_FOR
			END_IF
		ELSIF (cmd = M2C_NVI_UPDT_TOUT) THEN
			IF (unLastLen_mbxModule_1 = 3) THEN
				FOR z := 0 TO 1 DO
					IF aNviSnvtObjStatusIndex[z] = bNvRelativeIdx THEN
						paNviSnvtObjStatus[z]^.bStatusInformation.4 := BYTE_TO_BOOL(InDataTelegram_Module_1[2]);
						EXIT;
					END_IF
				END_FOR
			END_IF
		END_IF
	3, 19:
		IF (cmd = M2C_NVI_UPDT_OCCD) OR (cmd = M2C_NV_VALUE_RSP) THEN
			IF (unLastLen_mbxModule_1 = (2 + 29)) THEN
				FOR z := 0 TO 1 DO
					IF aNviSnvtAlarmIndex[z] = bNvRelativeIdx THEN
						FuRawToSnvtAlarm(ADR(InDataTelegram_Module_1[2]), paNviSnvtAlarm[z]);
						paNviSnvtAlarm[z]^.bInternalUseOnly.0 := FALSE;
						paNviSnvtAlarm[z]^.bStatusInformation := FuInkrementNviStatus(paNviSnvtAlarm[z]^.bStatusInformation);
						EXIT;
					END_IF
				END_FOR
			ELSIF (unLastLen_mbxModule_1 = 2) THEN
				FOR z := 0 TO 1 DO
					IF aNviSnvtAlarmIndex[z] = bNvRelativeIdx THEN
						paNviSnvtAlarm[z]^.bStatusInformation := FuInkrementNviStatus(paNviSnvtAlarm[z]^.bStatusInformation);
						EXIT;
					END_IF
				END_FOR
			END_IF
		ELSIF (cmd = M2C_NVI_UPDT_TOUT) THEN
			IF (unLastLen_mbxModule_1 = 3) THEN
				FOR z := 0 TO 1 DO
					IF aNviSnvtAlarmIndex[z] = bNvRelativeIdx THEN
						paNviSnvtAlarm[z]^.bStatusInformation.4 := BYTE_TO_BOOL(InDataTelegram_Module_1[2]);
						EXIT;
					END_IF
				END_FOR
			END_IF
		END_IF
	5, 21:
		IF (cmd = M2C_NVI_UPDT_OCCD) OR (cmd = M2C_NV_VALUE_RSP) THEN
			IF (unLastLen_mbxModule_1 = (2 + 2)) THEN
				FOR z := 0 TO 1 DO
					IF aNviSnvtStateIndex[z] = bNvRelativeIdx THEN
						FuRawToSnvtState(ADR(InDataTelegram_Module_1[2]), paNviSnvtState[z]);
						paNviSnvtState[z]^.bInternalUseOnly.0 := FALSE;
						paNviSnvtState[z]^.bStatusInformation := FuInkrementNviStatus(paNviSnvtState[z]^.bStatusInformation);
						EXIT;
					END_IF
				END_FOR
			ELSIF (unLastLen_mbxModule_1 = 2) THEN
				FOR z := 0 TO 1 DO
					IF aNviSnvtStateIndex[z] = bNvRelativeIdx THEN
						paNviSnvtState[z]^.bStatusInformation := FuInkrementNviStatus(paNviSnvtState[z]^.bStatusInformation);
						EXIT;
					END_IF
				END_FOR
			END_IF
		ELSIF (cmd = M2C_NVI_UPDT_TOUT) THEN
			IF (unLastLen_mbxModule_1 = 3) THEN
				FOR z := 0 TO 1 DO
					IF aNviSnvtStateIndex[z] = bNvRelativeIdx THEN
						paNviSnvtState[z]^.bStatusInformation.4 := BYTE_TO_BOOL(InDataTelegram_Module_1[2]);
						EXIT;
					END_IF
				END_FOR
			END_IF
		END_IF
	7, 9, 13, 15, 23, 25, 29, 31:
		IF (cmd = M2C_NVI_UPDT_OCCD) OR (cmd = M2C_NV_VALUE_RSP) THEN
			IF (unLastLen_mbxModule_1 = (2 + 2)) THEN
				FOR z := 0 TO 7 DO
					IF aNviSnvtTempPIndex[z] = bNvRelativeIdx THEN
						FuRawToSnvtTempP(ADR(InDataTelegram_Module_1[2]), paNviSnvtTempP[z]);
						paNviSnvtTempP[z]^.bInternalUseOnly.0 := FALSE;
						paNviSnvtTempP[z]^.bStatusInformation := FuInkrementNviStatus(paNviSnvtTempP[z]^.bStatusInformation);
						EXIT;
					END_IF
				END_FOR
			ELSIF (unLastLen_mbxModule_1 = 2) THEN
				FOR z := 0 TO 7 DO
					IF aNviSnvtTempPIndex[z] = bNvRelativeIdx THEN
						paNviSnvtTempP[z]^.bStatusInformation := FuInkrementNviStatus(paNviSnvtTempP[z]^.bStatusInformation);
						EXIT;
					END_IF
				END_FOR
			END_IF
		ELSIF (cmd = M2C_NVI_UPDT_TOUT) THEN
			IF (unLastLen_mbxModule_1 = 3) THEN
				FOR z := 0 TO 7 DO
					IF aNviSnvtTempPIndex[z] = bNvRelativeIdx THEN
						paNviSnvtTempP[z]^.bStatusInformation.4 := BYTE_TO_BOOL(InDataTelegram_Module_1[2]);
						EXIT;
					END_IF
				END_FOR
			END_IF
		END_IF
	11, 27:
		IF (cmd = M2C_NVI_UPDT_OCCD) OR (cmd = M2C_NV_VALUE_RSP) THEN
			IF (unLastLen_mbxModule_1 = (2 + 2)) THEN
				FOR z := 0 TO 1 DO
					IF aNviSnvtSwitchIndex[z] = bNvRelativeIdx THEN
						FuRawToSnvtSwitch(ADR(InDataTelegram_Module_1[2]), paNviSnvtSwitch[z]);
						paNviSnvtSwitch[z]^.bInternalUseOnly.0 := FALSE;
						paNviSnvtSwitch[z]^.bStatusInformation := FuInkrementNviStatus(paNviSnvtSwitch[z]^.bStatusInformation);
						EXIT;
					END_IF
				END_FOR
			ELSIF (unLastLen_mbxModule_1 = 2) THEN
				FOR z := 0 TO 1 DO
					IF aNviSnvtSwitchIndex[z] = bNvRelativeIdx THEN
						paNviSnvtSwitch[z]^.bStatusInformation := FuInkrementNviStatus(paNviSnvtSwitch[z]^.bStatusInformation);
						EXIT;
					END_IF
				END_FOR
			END_IF
		ELSIF (cmd = M2C_NVI_UPDT_TOUT) THEN
			IF (unLastLen_mbxModule_1 = 3) THEN
				FOR z := 0 TO 1 DO
					IF aNviSnvtSwitchIndex[z] = bNvRelativeIdx THEN
						paNviSnvtSwitch[z]^.bStatusInformation.4 := BYTE_TO_BOOL(InDataTelegram_Module_1[2]);
						EXIT;
					END_IF
				END_FOR
			END_IF
		END_IF

	END_CASE
ELSIF (cmd = M2C_CP_VALUE_RSP) THEN
	wCpRelativeIdx := ((InDataTelegram_Module_1[1] + InDataTelegram_Module_1[2] * 256) - wCpStartIndex - bObjectIndex) / bLmoCount;
	CASE wCpRelativeIdx OF

	END_CASE
END_IF
END_ACTION
ACTION ResetNviUpdate:
FOR z := 0 TO 1 DO
	paNviSnvtObjStatus[z]^.bStatusInformation := paNviSnvtObjStatus[z]^.bStatusInformation AND 16#F8;
END_FOR
FOR z := 0 TO 1 DO
	paNviSnvtAlarm[z]^.bStatusInformation := paNviSnvtAlarm[z]^.bStatusInformation AND 16#F8;
END_FOR
FOR z := 0 TO 1 DO
	paNviSnvtState[z]^.bStatusInformation := paNviSnvtState[z]^.bStatusInformation AND 16#F8;
END_FOR
FOR z := 0 TO 7 DO
	paNviSnvtTempP[z]^.bStatusInformation := paNviSnvtTempP[z]^.bStatusInformation AND 16#F8;
END_FOR
FOR z := 0 TO 1 DO
	paNviSnvtSwitch[z]^.bStatusInformation := paNviSnvtSwitch[z]^.bStatusInformation AND 16#F8;
END_FOR
;
END_ACTION
ACTION SendValueRequest:
FOR z := 0 TO 1 DO
	IF (FuSendNviValueReq_Module_1(ADR(paNviSnvtObjStatus[z]^.bInternalUseOnly), bNvStartIndex + bObjectIndex + (aNviSnvtObjStatusIndex[z] * bLmoCount)) = FALSE) THEN
		RETURN;
	END_IF;
END_FOR;
FOR z := 0 TO 1 DO
	IF (FuSendNviValueReq_Module_1(ADR(paNviSnvtAlarm[z]^.bInternalUseOnly), bNvStartIndex + bObjectIndex + (aNviSnvtAlarmIndex[z] * bLmoCount)) = FALSE) THEN
		RETURN;
	END_IF;
END_FOR;
FOR z := 0 TO 1 DO
	IF (FuSendNviValueReq_Module_1(ADR(paNviSnvtState[z]^.bInternalUseOnly), bNvStartIndex + bObjectIndex + (aNviSnvtStateIndex[z] * bLmoCount)) = FALSE) THEN
		RETURN;
	END_IF;
END_FOR;
FOR z := 0 TO 7 DO
	IF (FuSendNviValueReq_Module_1(ADR(paNviSnvtTempP[z]^.bInternalUseOnly), bNvStartIndex + bObjectIndex + (aNviSnvtTempPIndex[z] * bLmoCount)) = FALSE) THEN
		RETURN;
	END_IF;
END_FOR;
FOR z := 0 TO 1 DO
	IF (FuSendNviValueReq_Module_1(ADR(paNviSnvtSwitch[z]^.bInternalUseOnly), bNvStartIndex + bObjectIndex + (aNviSnvtSwitchIndex[z] * bLmoCount)) = FALSE) THEN
		RETURN;
	END_IF;
END_FOR;
;
END_ACTION
ACTION SetUpdateFlags:
FOR z := 0 TO 1 DO
	paNviSnvtObjStatus[z]^.bInternaluseOnly.0 := TRUE;
END_FOR;
FOR z := 0 TO 1 DO
	paNviSnvtAlarm[z]^.bInternaluseOnly.0 := TRUE;
END_FOR;
FOR z := 0 TO 1 DO
	paNviSnvtState[z]^.bInternaluseOnly.0 := TRUE;
END_FOR;
FOR z := 0 TO 7 DO
	paNviSnvtTempP[z]^.bInternaluseOnly.0 := TRUE;
END_FOR;
FOR z := 0 TO 1 DO
	paNviSnvtSwitch[z]^.bInternaluseOnly.0 := TRUE;
END_FOR;
FOR z := 0 TO 1 DO
	aNvoSnvtObjRequestLast[z].bInternaluseOnly.1 := TRUE;
	aNvoSnvtObjRequestLast[z].bInternaluseOnly.7 := (SHR(aNvoSnvtObjRequestPriority[z / 8], z MOD 8) AND 1) <> 0;
END_FOR;
FOR z := 0 TO 1 DO
	aNvoSnvtTimeStampLast[z].bInternaluseOnly.1 := TRUE;
	aNvoSnvtTimeStampLast[z].bInternaluseOnly.7 := (SHR(aNvoSnvtTimeStampPriority[z / 8], z MOD 8) AND 1) <> 0;
END_FOR;
FOR z := 0 TO 1 DO
	aNvoSnvtAlarmLast[z].bInternaluseOnly.1 := TRUE;
	aNvoSnvtAlarmLast[z].bInternaluseOnly.7 := (SHR(aNvoSnvtAlarmPriority[z / 8], z MOD 8) AND 1) <> 0;
END_FOR;
FOR z := 0 TO 3 DO
	aNvoSnvtHvacModeLast[z].bInternaluseOnly.1 := TRUE;
	aNvoSnvtHvacModeLast[z].bInternaluseOnly.7 := (SHR(aNvoSnvtHvacModePriority[z / 8], z MOD 8) AND 1) <> 0;
END_FOR;
FOR z := 0 TO 3 DO
	aNvoSnvtTempPLast[z].bInternaluseOnly.1 := TRUE;
	aNvoSnvtTempPLast[z].bInternaluseOnly.7 := (SHR(aNvoSnvtTempPPriority[z / 8], z MOD 8) AND 1) <> 0;
END_FOR;
FOR z := 0 TO 1 DO
	aNvoSnvtSwitchLast[z].bInternaluseOnly.1 := TRUE;
	aNvoSnvtSwitchLast[z].bInternaluseOnly.7 := (SHR(aNvoSnvtSwitchPriority[z / 8], z MOD 8) AND 1) <> 0;
END_FOR;
;
END_ACTION

(* POU LON/Shared/Internal/FuSnvtObjRequestToRaw, ST *)
FUNCTION FuSnvtObjRequestToRaw : BOOL
(******************************************)
(* Automatic generated code, do not edit! *)
(******************************************)
VAR_INPUT
	NvDataIn :  POINTER TO typSnvtObjRequest;
	DataOut : POINTER TO ARRAY[0..2] OF BYTE;
END_VAR
VAR
END_VAR
DataOut^[0] := WORD_TO_BYTE(SHR(NvDataIn^.wObjectId, 8));
DataOut^[1] := WORD_TO_BYTE(NvDataIn^.wObjectId);

DataOut^[2] := NvDataIn^.bObjectRequest;

FuSnvtObjRequestToRaw := TRUE;
END_FUNCTION

